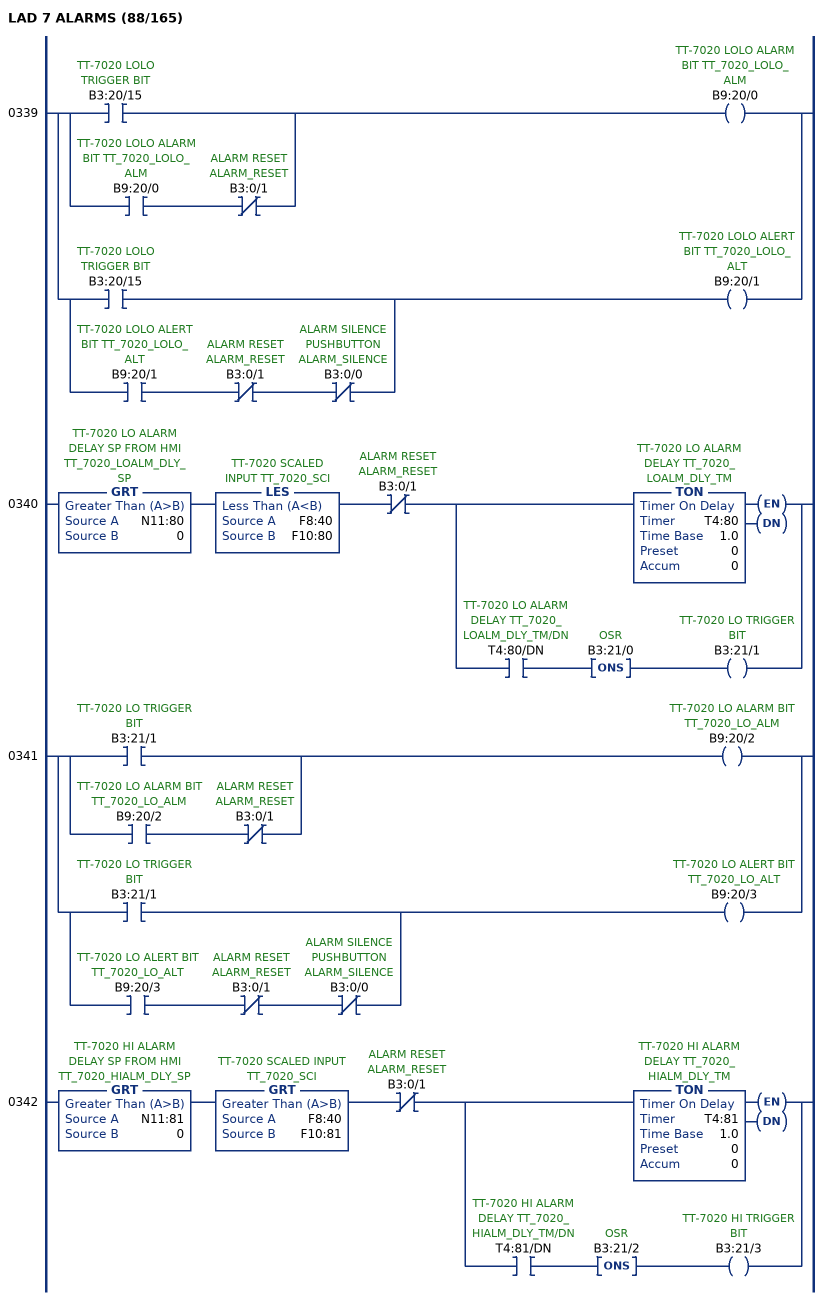
% Rung: 339 %
SOR BST BST XIC B3:20/15 NXB XIC B9:20/0 XIO B3:0/1 BND OTE B9:20/0 NXB BST XIC B3:20/15 NXB XIC B9:20/1 XIO B3:0/1 XIO B3:0/0 BND OTE B9:20/1 BND EOR
%   B3:20/15  "TT-7020 LOLO TRIGGER BIT" %
%   B9:20/0  TT_7020_LOLO_ALM  "TT-7020 LOLO ALARM BIT" %
%   B3:0/1  ALARM_RESET  "ALARM RESET" %
%   B9:20/1  TT_7020_LOLO_ALT  "TT-7020 LOLO ALERT BIT" %
%   B3:0/0  ALARM_SILENCE  "ALARM SILENCE PUSHBUTTON" %
% Rung: 340 %
SOR GRT N11:80 0 LES F8:40 F10:80 XIO B3:0/1 BST TON T4:80 1.0 0 0 NXB XIC T4:80/DN OSR B3:21/0 OTE B3:21/1 BND EOR
%   N11:80  TT_7020_LOALM_DLY_SP  "TT-7020 LO ALARM DELAY SP FROM HMI" %
%   F8:40  TT_7020_SCI  "TT-7020 SCALED INPUT" %
%   F10:80  TT_7020_LOALM_SP  "TT-7020 LO ALARM SP" %
%   B3:0/1  ALARM_RESET  "ALARM RESET" %
%   T4:80  TT_7020_LOALM_DLY_TM  "TT-7020 LO ALARM DELAY" %
%   B3:21/0  "OSR" %
%   B3:21/1  "TT-7020 LO TRIGGER BIT" %
% Rung: 341 %
SOR BST BST XIC B3:21/1 NXB XIC B9:20/2 XIO B3:0/1 BND OTE B9:20/2 NXB BST XIC B3:21/1 NXB XIC B9:20/3 XIO B3:0/1 XIO B3:0/0 BND OTE B9:20/3 BND EOR
%   B3:21/1  "TT-7020 LO TRIGGER BIT" %
%   B9:20/2  TT_7020_LO_ALM  "TT-7020 LO ALARM BIT" %
%   B3:0/1  ALARM_RESET  "ALARM RESET" %
%   B9:20/3  TT_7020_LO_ALT  "TT-7020 LO ALERT BIT" %
%   B3:0/0  ALARM_SILENCE  "ALARM SILENCE PUSHBUTTON" %
% Rung: 342 %
SOR GRT N11:81 0 GRT F8:40 F10:81 XIO B3:0/1 BST TON T4:81 1.0 0 0 NXB XIC T4:81/DN OSR B3:21/2 OTE B3:21/3 BND EOR
%   N11:81  TT_7020_HIALM_DLY_SP  "TT-7020 HI ALARM DELAY SP FROM HMI" %
%   F8:40  TT_7020_SCI  "TT-7020 SCALED INPUT" %
%   F10:81  TT_7020_HIALM_SP  "TT-7020 HI ALARM SP" %
%   B3:0/1  ALARM_RESET  "ALARM RESET" %
%   T4:81  TT_7020_HIALM_DLY_TM  "TT-7020 HI ALARM DELAY" %
%   B3:21/2  "OSR" %
%   B3:21/3  "TT-7020 HI TRIGGER BIT" %

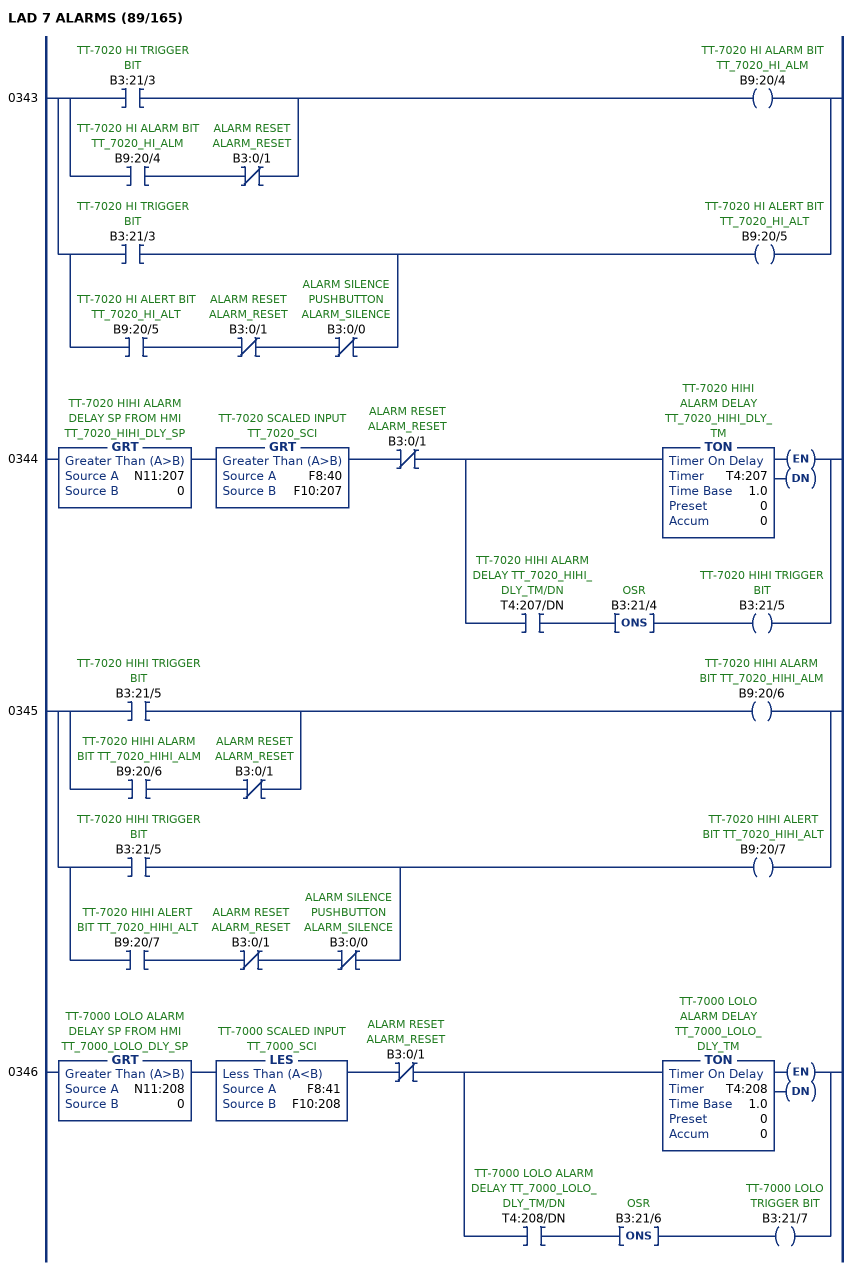
% Rung: 343 %
SOR BST BST XIC B3:21/3 NXB XIC B9:20/4 XIO B3:0/1 BND OTE B9:20/4 NXB BST XIC B3:21/3 NXB XIC B9:20/5 XIO B3:0/1 XIO B3:0/0 BND OTE B9:20/5 BND EOR
%   B3:21/3  "TT-7020 HI TRIGGER BIT" %
%   B9:20/4  TT_7020_HI_ALM  "TT-7020 HI ALARM BIT" %
%   B3:0/1  ALARM_RESET  "ALARM RESET" %
%   B9:20/5  TT_7020_HI_ALT  "TT-7020 HI ALERT BIT" %
%   B3:0/0  ALARM_SILENCE  "ALARM SILENCE PUSHBUTTON" %
% Rung: 344 %
SOR GRT N11:207 0 GRT F8:40 F10:207 XIO B3:0/1 BST TON T4:207 1.0 0 0 NXB XIC T4:207/DN OSR B3:21/4 OTE B3:21/5 BND EOR
%   N11:207  TT_7020_HIHI_DLY_SP  "TT-7020 HIHI ALARM DELAY SP FROM HMI" %
%   F8:40  TT_7020_SCI  "TT-7020 SCALED INPUT" %
%   F10:207  TT_7020_HIHI_SP  "TT-7020 HIHI ALARM SP" %
%   B3:0/1  ALARM_RESET  "ALARM RESET" %
%   T4:207  TT_7020_HIHI_DLY_TM  "TT-7020 HIHI ALARM DELAY" %
%   B3:21/4  "OSR" %
%   B3:21/5  "TT-7020 HIHI TRIGGER BIT" %
% Rung: 345 %
SOR BST BST XIC B3:21/5 NXB XIC B9:20/6 XIO B3:0/1 BND OTE B9:20/6 NXB BST XIC B3:21/5 NXB XIC B9:20/7 XIO B3:0/1 XIO B3:0/0 BND OTE B9:20/7 BND EOR
%   B3:21/5  "TT-7020 HIHI TRIGGER BIT" %
%   B9:20/6  TT_7020_HIHI_ALM  "TT-7020 HIHI ALARM BIT" %
%   B3:0/1  ALARM_RESET  "ALARM RESET" %
%   B9:20/7  TT_7020_HIHI_ALT  "TT-7020 HIHI ALERT BIT" %
%   B3:0/0  ALARM_SILENCE  "ALARM SILENCE PUSHBUTTON" %
% Rung: 346 %
SOR GRT N11:208 0 LES F8:41 F10:208 XIO B3:0/1 BST TON T4:208 1.0 0 0 NXB XIC T4:208/DN OSR B3:21/6 OTE B3:21/7 BND EOR
%   N11:208  TT_7000_LOLO_DLY_SP  "TT-7000 LOLO ALARM DELAY SP FROM HMI" %
%   F8:41  TT_7000_SCI  "TT-7000 SCALED INPUT" %
%   F10:208  TT_7000_LOLO_SP  "TT-7000 LOLO ALARM SP" %
%   B3:0/1  ALARM_RESET  "ALARM RESET" %
%   T4:208  TT_7000_LOLO_DLY_TM  "TT-7000 LOLO ALARM DELAY" %
%   B3:21/6  "OSR" %
%   B3:21/7  "TT-7000 LOLO TRIGGER BIT" %

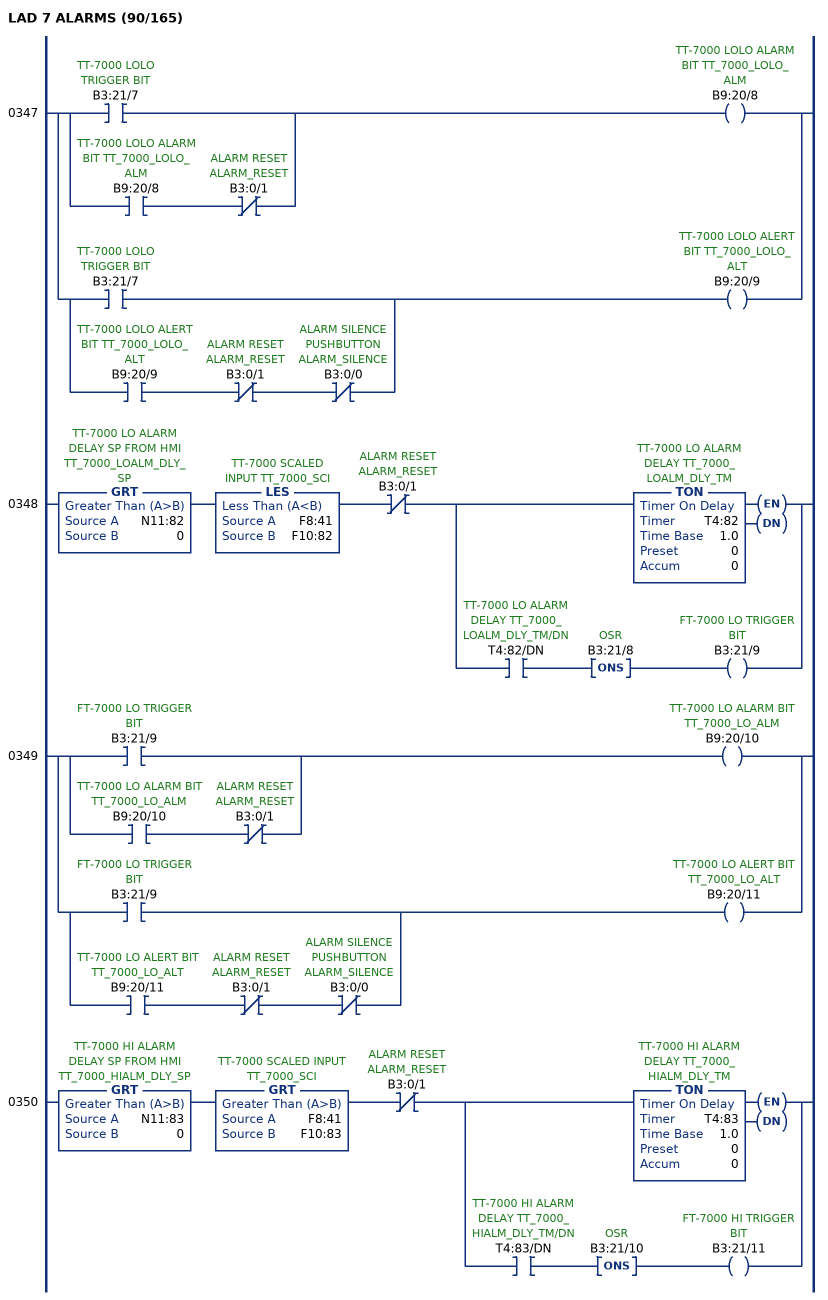
% Rung: 347 %
SOR BST BST XIC B3:21/7 NXB XIC B9:20/8 XIO B3:0/1 BND OTE B9:20/8 NXB BST XIC B3:21/7 NXB XIC B9:20/9 XIO B3:0/1 XIO B3:0/0 BND OTE B9:20/9 BND EOR
%   B3:21/7  "TT-7000 LOLO TRIGGER BIT" %
%   B9:20/8  TT_7000_LOLO_ALM  "TT-7000 LOLO ALARM BIT" %
%   B3:0/1  ALARM_RESET  "ALARM RESET" %
%   B9:20/9  TT_7000_LOLO_ALT  "TT-7000 LOLO ALERT BIT" %
%   B3:0/0  ALARM_SILENCE  "ALARM SILENCE PUSHBUTTON" %
% Rung: 348 %
SOR GRT N11:82 0 LES F8:41 F10:82 XIO B3:0/1 BST TON T4:82 1.0 0 0 NXB XIC T4:82/DN OSR B3:21/8 OTE B3:21/9 BND EOR
%   N11:82  TT_7000_LOALM_DLY_SP  "TT-7000 LO ALARM DELAY SP FROM HMI" %
%   F8:41  TT_7000_SCI  "TT-7000 SCALED INPUT" %
%   F10:82  TT_7000_LOALM_SP  "TT-7000 LO ALARM SP" %
%   B3:0/1  ALARM_RESET  "ALARM RESET" %
%   T4:82  TT_7000_LOALM_DLY_TM  "TT-7000 LO ALARM DELAY" %
%   B3:21/8  "OSR" %
%   B3:21/9  "FT-7000 LO TRIGGER BIT" %
% Rung: 349 %
SOR BST BST XIC B3:21/9 NXB XIC B9:20/10 XIO B3:0/1 BND OTE B9:20/10 NXB BST XIC B3:21/9 NXB XIC B9:20/11 XIO B3:0/1 XIO B3:0/0 BND OTE B9:20/11 BND EOR
%   B3:21/9  "FT-7000 LO TRIGGER BIT" %
%   B9:20/10  TT_7000_LO_ALM  "TT-7000 LO ALARM BIT" %
%   B3:0/1  ALARM_RESET  "ALARM RESET" %
%   B9:20/11  TT_7000_LO_ALT  "TT-7000 LO ALERT BIT" %
%   B3:0/0  ALARM_SILENCE  "ALARM SILENCE PUSHBUTTON" %
% Rung: 350 %
SOR GRT N11:83 0 GRT F8:41 F10:83 XIO B3:0/1 BST TON T4:83 1.0 0 0 NXB XIC T4:83/DN OSR B3:21/10 OTE B3:21/11 BND EOR
%   N11:83  TT_7000_HIALM_DLY_SP  "TT-7000 HI ALARM DELAY SP FROM HMI" %
%   F8:41  TT_7000_SCI  "TT-7000 SCALED INPUT" %
%   F10:83  TT_7000_HIALM_SP  "TT-7000 HI ALARM SP" %
%   B3:0/1  ALARM_RESET  "ALARM RESET" %
%   T4:83  TT_7000_HIALM_DLY_TM  "TT-7000 HI ALARM DELAY" %
%   B3:21/10  "OSR" %
%   B3:21/11  "FT-7000 HI TRIGGER BIT" %

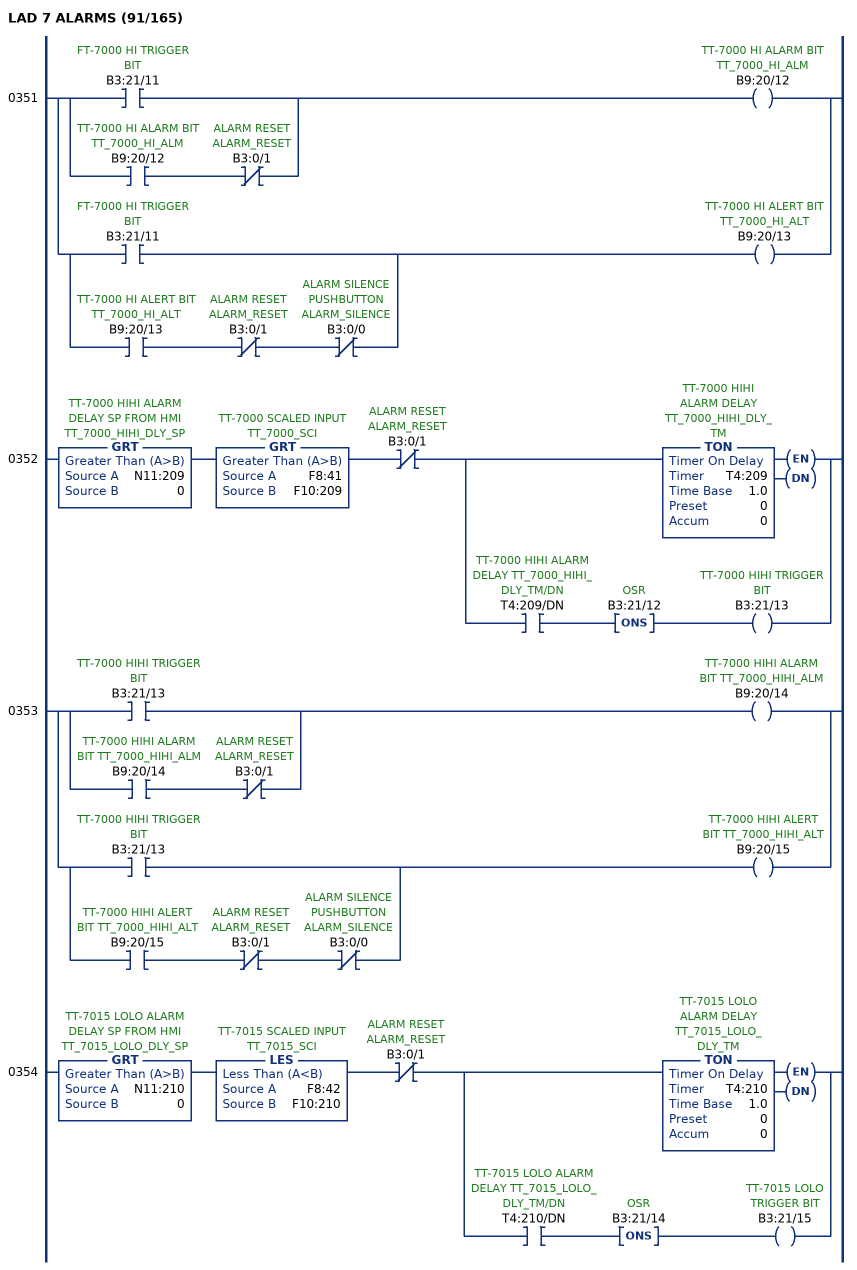
% Rung: 351 %
SOR BST BST XIC B3:21/11 NXB XIC B9:20/12 XIO B3:0/1 BND OTE B9:20/12 NXB BST XIC B3:21/11 NXB XIC B9:20/13 XIO B3:0/1 XIO B3:0/0 BND OTE B9:20/13 BND EOR
%   B3:21/11  "FT-7000 HI TRIGGER BIT" %
%   B9:20/12  TT_7000_HI_ALM  "TT-7000 HI ALARM BIT" %
%   B3:0/1  ALARM_RESET  "ALARM RESET" %
%   B9:20/13  TT_7000_HI_ALT  "TT-7000 HI ALERT BIT" %
%   B3:0/0  ALARM_SILENCE  "ALARM SILENCE PUSHBUTTON" %
% Rung: 352 %
SOR GRT N11:209 0 GRT F8:41 F10:209 XIO B3:0/1 BST TON T4:209 1.0 0 0 NXB XIC T4:209/DN OSR B3:21/12 OTE B3:21/13 BND EOR
%   N11:209  TT_7000_HIHI_DLY_SP  "TT-7000 HIHI ALARM DELAY SP FROM HMI" %
%   F8:41  TT_7000_SCI  "TT-7000 SCALED INPUT" %
%   F10:209  TT_7000_HIHI_SP  "TT-7000 HIHI ALARM SP" %
%   B3:0/1  ALARM_RESET  "ALARM RESET" %
%   T4:209  TT_7000_HIHI_DLY_TM  "TT-7000 HIHI ALARM DELAY" %
%   B3:21/12  "OSR" %
%   B3:21/13  "TT-7000 HIHI TRIGGER BIT" %
% Rung: 353 %
SOR BST BST XIC B3:21/13 NXB XIC B9:20/14 XIO B3:0/1 BND OTE B9:20/14 NXB BST XIC B3:21/13 NXB XIC B9:20/15 XIO B3:0/1 XIO B3:0/0 BND OTE B9:20/15 BND EOR
%   B3:21/13  "TT-7000 HIHI TRIGGER BIT" %
%   B9:20/14  TT_7000_HIHI_ALM  "TT-7000 HIHI ALARM BIT" %
%   B3:0/1  ALARM_RESET  "ALARM RESET" %
%   B9:20/15  TT_7000_HIHI_ALT  "TT-7000 HIHI ALERT BIT" %
%   B3:0/0  ALARM_SILENCE  "ALARM SILENCE PUSHBUTTON" %
% Rung: 354 %
SOR GRT N11:210 0 LES F8:42 F10:210 XIO B3:0/1 BST TON T4:210 1.0 0 0 NXB XIC T4:210/DN OSR B3:21/14 OTE B3:21/15 BND EOR
%   N11:210  TT_7015_LOLO_DLY_SP  "TT-7015 LOLO ALARM DELAY SP FROM HMI" %
%   F8:42  TT_7015_SCI  "TT-7015 SCALED INPUT" %
%   F10:210  TT_7015_LOLO_SP  "TT-7015 LOLO ALARM SP" %
%   B3:0/1  ALARM_RESET  "ALARM RESET" %
%   T4:210  TT_7015_LOLO_DLY_TM  "TT-7015 LOLO ALARM DELAY" %
%   B3:21/14  "OSR" %
%   B3:21/15  "TT-7015 LOLO TRIGGER BIT" %

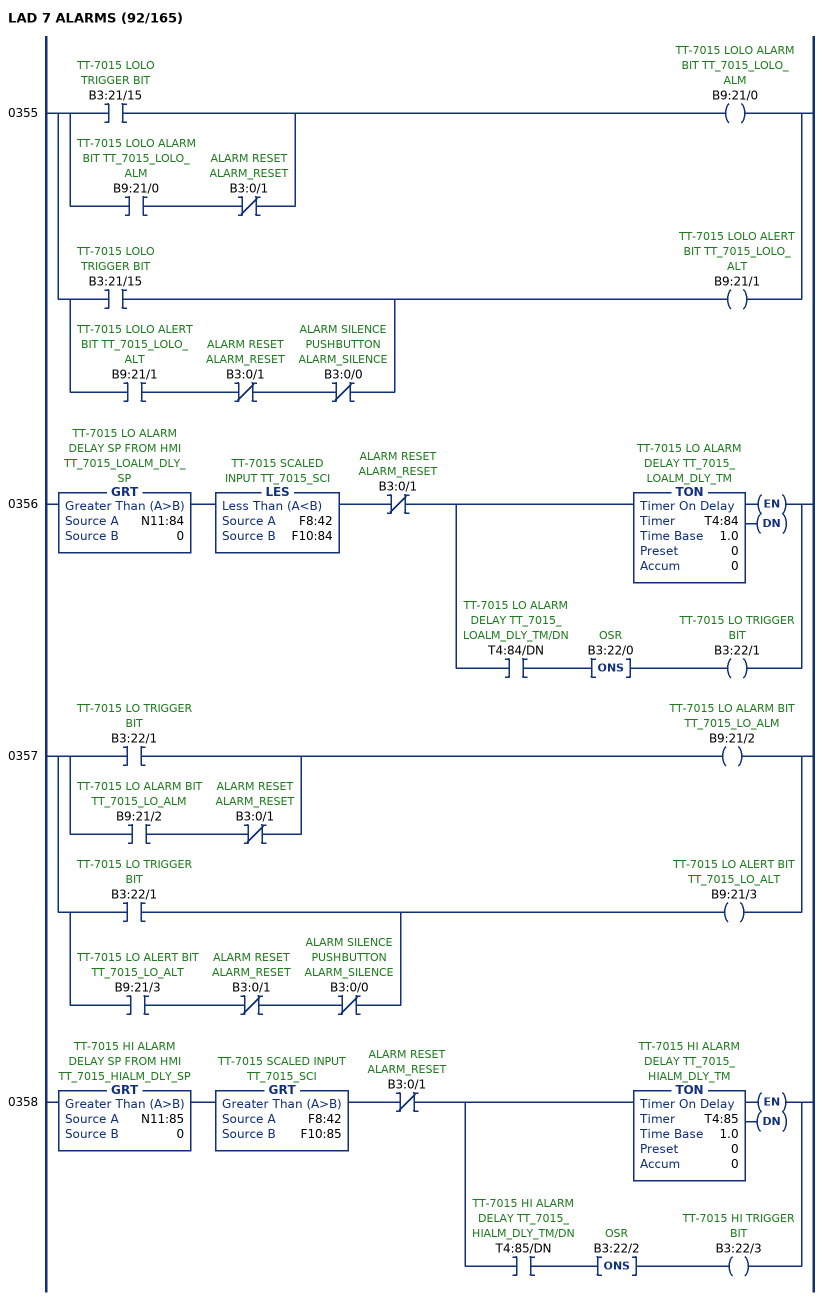
% Rung: 355 %
SOR BST BST XIC B3:21/15 NXB XIC B9:21/0 XIO B3:0/1 BND OTE B9:21/0 NXB BST XIC B3:21/15 NXB XIC B9:21/1 XIO B3:0/1 XIO B3:0/0 BND OTE B9:21/1 BND EOR
%   B3:21/15  "TT-7015 LOLO TRIGGER BIT" %
%   B9:21/0  TT_7015_LOLO_ALM  "TT-7015 LOLO ALARM BIT" %
%   B3:0/1  ALARM_RESET  "ALARM RESET" %
%   B9:21/1  TT_7015_LOLO_ALT  "TT-7015 LOLO ALERT BIT" %
%   B3:0/0  ALARM_SILENCE  "ALARM SILENCE PUSHBUTTON" %
% Rung: 356 %
SOR GRT N11:84 0 LES F8:42 F10:84 XIO B3:0/1 BST TON T4:84 1.0 0 0 NXB XIC T4:84/DN OSR B3:22/0 OTE B3:22/1 BND EOR
%   N11:84  TT_7015_LOALM_DLY_SP  "TT-7015 LO ALARM DELAY SP FROM HMI" %
%   F8:42  TT_7015_SCI  "TT-7015 SCALED INPUT" %
%   F10:84  TT_7015_LOALM_SP  "TT-7015 LO ALARM SP" %
%   B3:0/1  ALARM_RESET  "ALARM RESET" %
%   T4:84  TT_7015_LOALM_DLY_TM  "TT-7015 LO ALARM DELAY" %
%   B3:22/0  "OSR" %
%   B3:22/1  "TT-7015 LO TRIGGER BIT" %
% Rung: 357 %
SOR BST BST XIC B3:22/1 NXB XIC B9:21/2 XIO B3:0/1 BND OTE B9:21/2 NXB BST XIC B3:22/1 NXB XIC B9:21/3 XIO B3:0/1 XIO B3:0/0 BND OTE B9:21/3 BND EOR
%   B3:22/1  "TT-7015 LO TRIGGER BIT" %
%   B9:21/2  TT_7015_LO_ALM  "TT-7015 LO ALARM BIT" %
%   B3:0/1  ALARM_RESET  "ALARM RESET" %
%   B9:21/3  TT_7015_LO_ALT  "TT-7015 LO ALERT BIT" %
%   B3:0/0  ALARM_SILENCE  "ALARM SILENCE PUSHBUTTON" %
% Rung: 358 %
SOR GRT N11:85 0 GRT F8:42 F10:85 XIO B3:0/1 BST TON T4:85 1.0 0 0 NXB XIC T4:85/DN OSR B3:22/2 OTE B3:22/3 BND EOR
%   N11:85  TT_7015_HIALM_DLY_SP  "TT-7015 HI ALARM DELAY SP FROM HMI" %
%   F8:42  TT_7015_SCI  "TT-7015 SCALED INPUT" %
%   F10:85  TT_7015_HIALM_SP  "TT-7015 HI ALARM SP" %
%   B3:0/1  ALARM_RESET  "ALARM RESET" %
%   T4:85  TT_7015_HIALM_DLY_TM  "TT-7015 HI ALARM DELAY" %
%   B3:22/2  "OSR" %
%   B3:22/3  "TT-7015 HI TRIGGER BIT" %

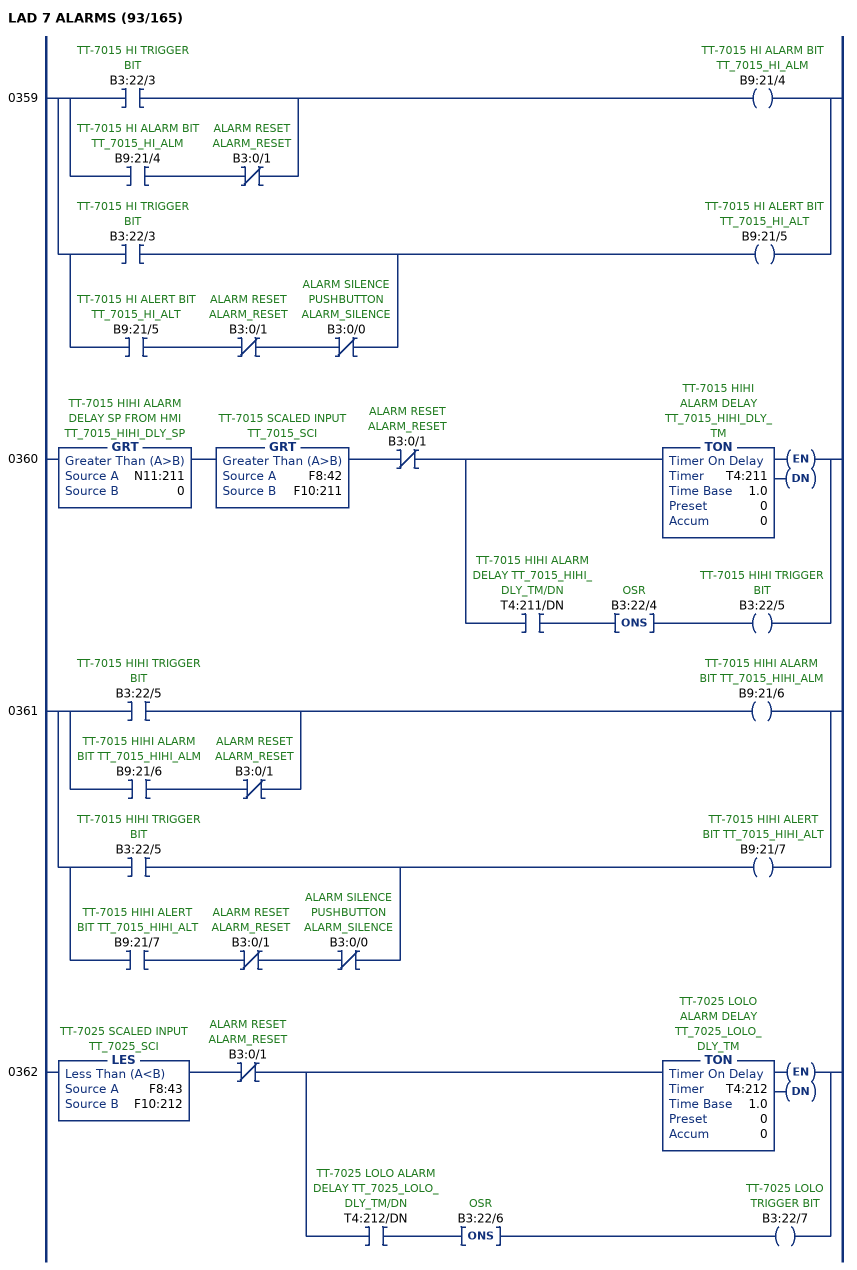
% Rung: 359 %
SOR BST BST XIC B3:22/3 NXB XIC B9:21/4 XIO B3:0/1 BND OTE B9:21/4 NXB BST XIC B3:22/3 NXB XIC B9:21/5 XIO B3:0/1 XIO B3:0/0 BND OTE B9:21/5 BND EOR
%   B3:22/3  "TT-7015 HI TRIGGER BIT" %
%   B9:21/4  TT_7015_HI_ALM  "TT-7015 HI ALARM BIT" %
%   B3:0/1  ALARM_RESET  "ALARM RESET" %
%   B9:21/5  TT_7015_HI_ALT  "TT-7015 HI ALERT BIT" %
%   B3:0/0  ALARM_SILENCE  "ALARM SILENCE PUSHBUTTON" %
% Rung: 360 %
SOR GRT N11:211 0 GRT F8:42 F10:211 XIO B3:0/1 BST TON T4:211 1.0 0 0 NXB XIC T4:211/DN OSR B3:22/4 OTE B3:22/5 BND EOR
%   N11:211  TT_7015_HIHI_DLY_SP  "TT-7015 HIHI ALARM DELAY SP FROM HMI" %
%   F8:42  TT_7015_SCI  "TT-7015 SCALED INPUT" %
%   F10:211  TT_7015_HIHI_SP  "TT-7015 HIHI ALARM SP" %
%   B3:0/1  ALARM_RESET  "ALARM RESET" %
%   T4:211  TT_7015_HIHI_DLY_TM  "TT-7015 HIHI ALARM DELAY" %
%   B3:22/4  "OSR" %
%   B3:22/5  "TT-7015 HIHI TRIGGER BIT" %
% Rung: 361 %
SOR BST BST XIC B3:22/5 NXB XIC B9:21/6 XIO B3:0/1 BND OTE B9:21/6 NXB BST XIC B3:22/5 NXB XIC B9:21/7 XIO B3:0/1 XIO B3:0/0 BND OTE B9:21/7 BND EOR
%   B3:22/5  "TT-7015 HIHI TRIGGER BIT" %
%   B9:21/6  TT_7015_HIHI_ALM  "TT-7015 HIHI ALARM BIT" %
%   B3:0/1  ALARM_RESET  "ALARM RESET" %
%   B9:21/7  TT_7015_HIHI_ALT  "TT-7015 HIHI ALERT BIT" %
%   B3:0/0  ALARM_SILENCE  "ALARM SILENCE PUSHBUTTON" %
% Rung: 362 %
SOR LES F8:43 F10:212 XIO B3:0/1 BST TON T4:212 1.0 0 0 NXB XIC T4:212/DN OSR B3:22/6 OTE B3:22/7 BND EOR
%   F8:43  TT_7025_SCI  "TT-7025 SCALED INPUT" %
%   F10:212  TT_7025_LOLO_SP  "TT-7025 LOLO ALARM SP" %
%   B3:0/1  ALARM_RESET  "ALARM RESET" %
%   T4:212  TT_7025_LOLO_DLY_TM  "TT-7025 LOLO ALARM DELAY" %
%   B3:22/6  "OSR" %
%   B3:22/7  "TT-7025 LOLO TRIGGER BIT" %

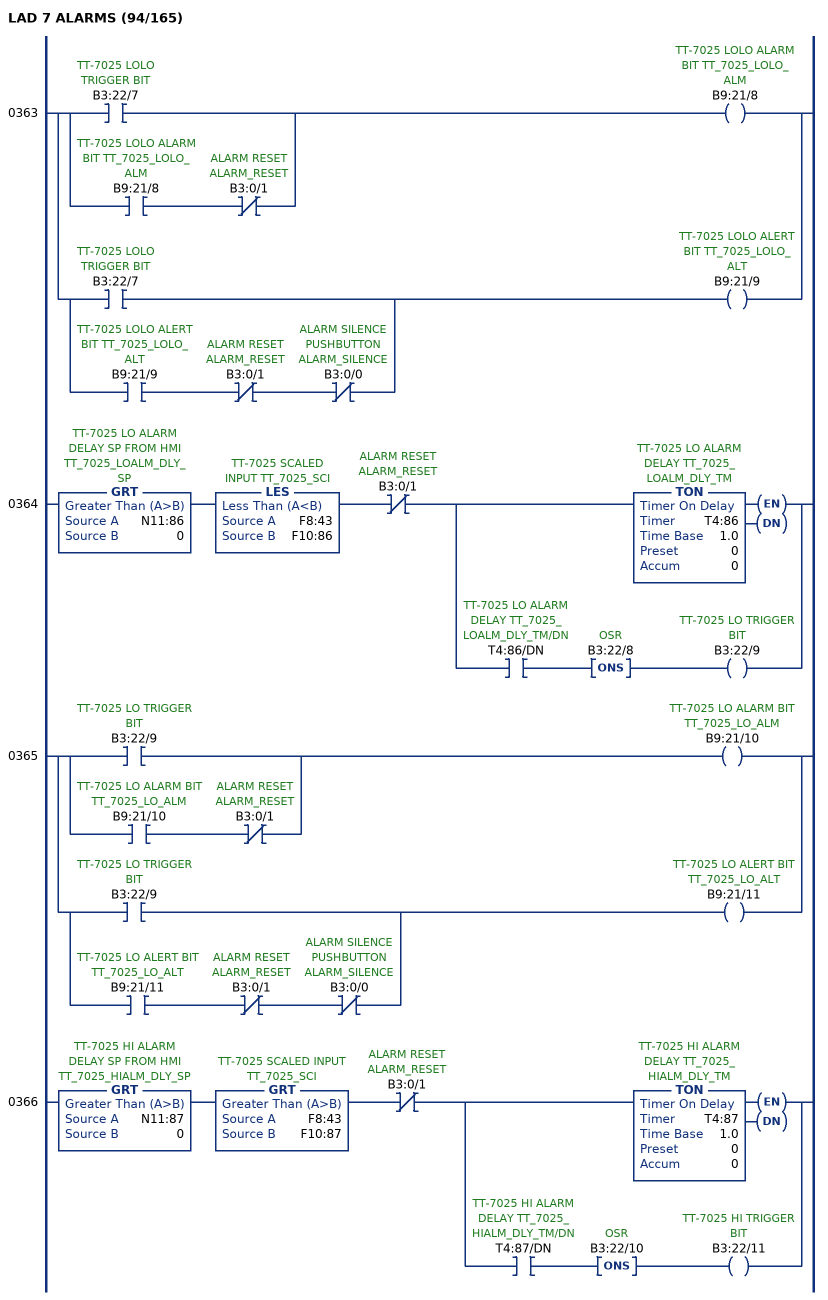
% Rung: 363 %
SOR BST BST XIC B3:22/7 NXB XIC B9:21/8 XIO B3:0/1 BND OTE B9:21/8 NXB BST XIC B3:22/7 NXB XIC B9:21/9 XIO B3:0/1 XIO B3:0/0 BND OTE B9:21/9 BND EOR
%   B3:22/7  "TT-7025 LOLO TRIGGER BIT" %
%   B9:21/8  TT_7025_LOLO_ALM  "TT-7025 LOLO ALARM BIT" %
%   B3:0/1  ALARM_RESET  "ALARM RESET" %
%   B9:21/9  TT_7025_LOLO_ALT  "TT-7025 LOLO ALERT BIT" %
%   B3:0/0  ALARM_SILENCE  "ALARM SILENCE PUSHBUTTON" %
% Rung: 364 %
SOR GRT N11:86 0 LES F8:43 F10:86 XIO B3:0/1 BST TON T4:86 1.0 0 0 NXB XIC T4:86/DN OSR B3:22/8 OTE B3:22/9 BND EOR
%   N11:86  TT_7025_LOALM_DLY_SP  "TT-7025 LO ALARM DELAY SP FROM HMI" %
%   F8:43  TT_7025_SCI  "TT-7025 SCALED INPUT" %
%   F10:86  TT_7025_LOALM_SP  "TT-7025 LO ALARM SP" %
%   B3:0/1  ALARM_RESET  "ALARM RESET" %
%   T4:86  TT_7025_LOALM_DLY_TM  "TT-7025 LO ALARM DELAY" %
%   B3:22/8  "OSR" %
%   B3:22/9  "TT-7025 LO TRIGGER BIT" %
% Rung: 365 %
SOR BST BST XIC B3:22/9 NXB XIC B9:21/10 XIO B3:0/1 BND OTE B9:21/10 NXB BST XIC B3:22/9 NXB XIC B9:21/11 XIO B3:0/1 XIO B3:0/0 BND OTE B9:21/11 BND EOR
%   B3:22/9  "TT-7025 LO TRIGGER BIT" %
%   B9:21/10  TT_7025_LO_ALM  "TT-7025 LO ALARM BIT" %
%   B3:0/1  ALARM_RESET  "ALARM RESET" %
%   B9:21/11  TT_7025_LO_ALT  "TT-7025 LO ALERT BIT" %
%   B3:0/0  ALARM_SILENCE  "ALARM SILENCE PUSHBUTTON" %
% Rung: 366 %
SOR GRT N11:87 0 GRT F8:43 F10:87 XIO B3:0/1 BST TON T4:87 1.0 0 0 NXB XIC T4:87/DN OSR B3:22/10 OTE B3:22/11 BND EOR
%   N11:87  TT_7025_HIALM_DLY_SP  "TT-7025 HI ALARM DELAY SP FROM HMI" %
%   F8:43  TT_7025_SCI  "TT-7025 SCALED INPUT" %
%   F10:87  TT_7025_HIALM_SP  "TT-7025 HI ALARM SP" %
%   B3:0/1  ALARM_RESET  "ALARM RESET" %
%   T4:87  TT_7025_HIALM_DLY_TM  "TT-7025 HI ALARM DELAY" %
%   B3:22/10  "OSR" %
%   B3:22/11  "TT-7025 HI TRIGGER BIT" %

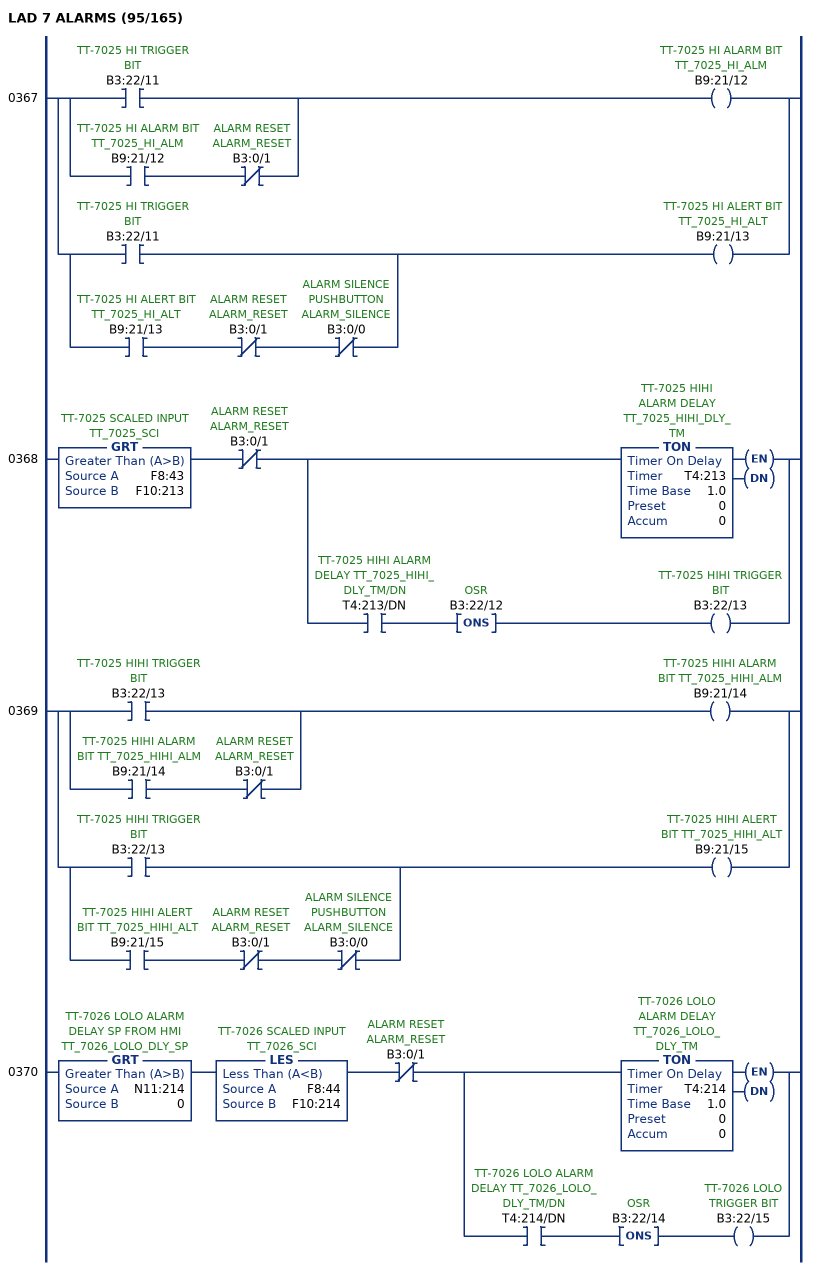
% Rung: 367 %
SOR BST BST XIC B3:22/11 NXB XIC B9:21/12 XIO B3:0/1 BND OTE B9:21/12 NXB BST XIC B3:22/11 NXB XIC B9:21/13 XIO B3:0/1 XIO B3:0/0 BND OTE B9:21/13 BND EOR
%   B3:22/11  "TT-7025 HI TRIGGER BIT" %
%   B9:21/12  TT_7025_HI_ALM  "TT-7025 HI ALARM BIT" %
%   B3:0/1  ALARM_RESET  "ALARM RESET" %
%   B9:21/13  TT_7025_HI_ALT  "TT-7025 HI ALERT BIT" %
%   B3:0/0  ALARM_SILENCE  "ALARM SILENCE PUSHBUTTON" %
% Rung: 368 %
SOR GRT F8:43 F10:213 XIO B3:0/1 BST TON T4:213 1.0 0 0 NXB XIC T4:213/DN OSR B3:22/12 OTE B3:22/13 BND EOR
%   F8:43  TT_7025_SCI  "TT-7025 SCALED INPUT" %
%   F10:213  TT_7025_HIHI_SP  "TT-7025 HIHI ALARM SP" %
%   B3:0/1  ALARM_RESET  "ALARM RESET" %
%   T4:213  TT_7025_HIHI_DLY_TM  "TT-7025 HIHI ALARM DELAY" %
%   B3:22/12  "OSR" %
%   B3:22/13  "TT-7025 HIHI TRIGGER BIT" %
% Rung: 369 %
SOR BST BST XIC B3:22/13 NXB XIC B9:21/14 XIO B3:0/1 BND OTE B9:21/14 NXB BST XIC B3:22/13 NXB XIC B9:21/15 XIO B3:0/1 XIO B3:0/0 BND OTE B9:21/15 BND EOR
%   B3:22/13  "TT-7025 HIHI TRIGGER BIT" %
%   B9:21/14  TT_7025_HIHI_ALM  "TT-7025 HIHI ALARM BIT" %
%   B3:0/1  ALARM_RESET  "ALARM RESET" %
%   B9:21/15  TT_7025_HIHI_ALT  "TT-7025 HIHI ALERT BIT" %
%   B3:0/0  ALARM_SILENCE  "ALARM SILENCE PUSHBUTTON" %
% Rung: 370 %
SOR GRT N11:214 0 LES F8:44 F10:214 XIO B3:0/1 BST TON T4:214 1.0 0 0 NXB XIC T4:214/DN OSR B3:22/14 OTE B3:22/15 BND EOR
%   N11:214  TT_7026_LOLO_DLY_SP  "TT-7026 LOLO ALARM DELAY SP FROM HMI" %
%   F8:44  TT_7026_SCI  "TT-7026 SCALED INPUT" %
%   F10:214  TT_7026_LOLO_SP  "TT-7026 LOLO ALARM SP" %
%   B3:0/1  ALARM_RESET  "ALARM RESET" %
%   T4:214  TT_7026_LOLO_DLY_TM  "TT-7026 LOLO ALARM DELAY" %
%   B3:22/14  "OSR" %
%   B3:22/15  "TT-7026 LOLO TRIGGER BIT" %

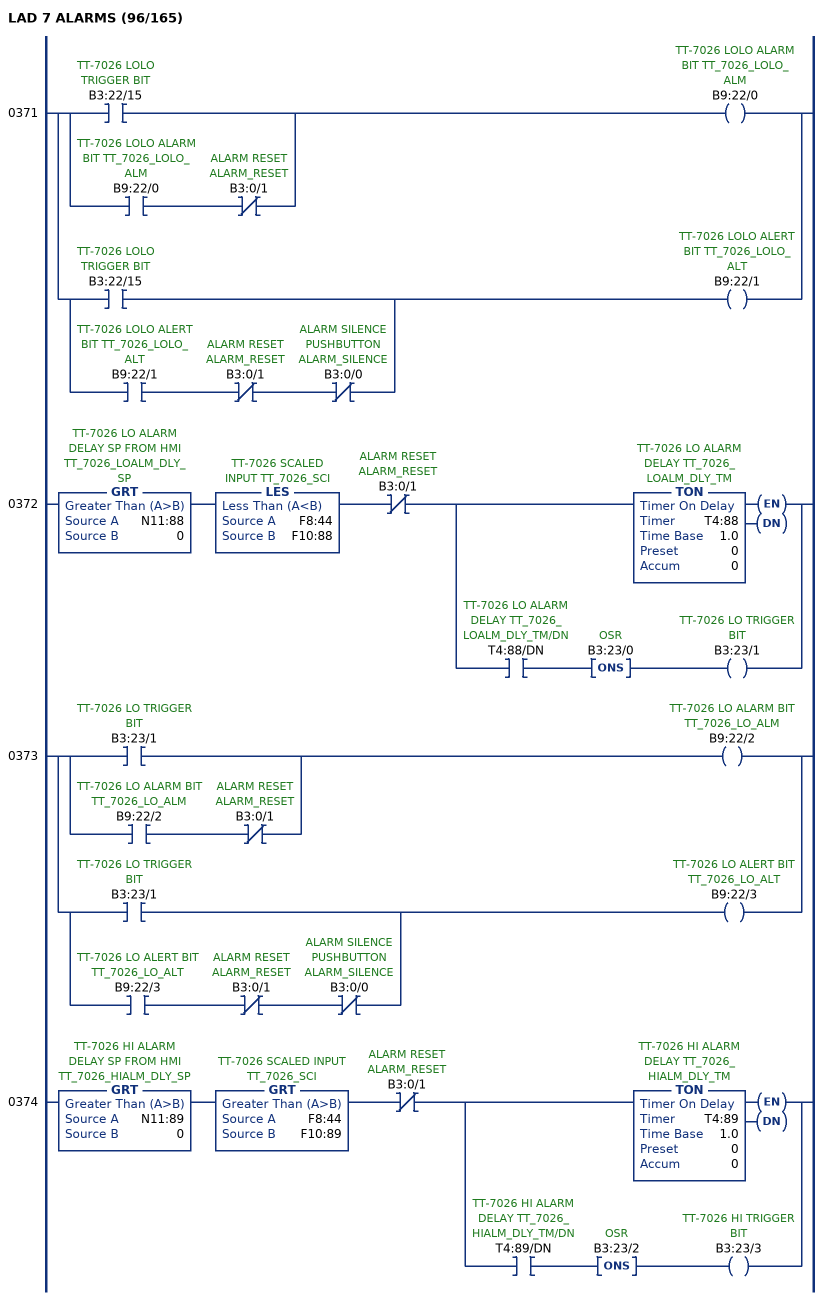
% Rung: 371 %
SOR BST BST XIC B3:22/15 NXB XIC B9:22/0 XIO B3:0/1 BND OTE B9:22/0 NXB BST XIC B3:22/15 NXB XIC B9:22/1 XIO B3:0/1 XIO B3:0/0 BND OTE B9:22/1 BND EOR
%   B3:22/15  "TT-7026 LOLO TRIGGER BIT" %
%   B9:22/0  TT_7026_LOLO_ALM  "TT-7026 LOLO ALARM BIT" %
%   B3:0/1  ALARM_RESET  "ALARM RESET" %
%   B9:22/1  TT_7026_LOLO_ALT  "TT-7026 LOLO ALERT BIT" %
%   B3:0/0  ALARM_SILENCE  "ALARM SILENCE PUSHBUTTON" %
% Rung: 372 %
SOR GRT N11:88 0 LES F8:44 F10:88 XIO B3:0/1 BST TON T4:88 1.0 0 0 NXB XIC T4:88/DN OSR B3:23/0 OTE B3:23/1 BND EOR
%   N11:88  TT_7026_LOALM_DLY_SP  "TT-7026 LO ALARM DELAY SP FROM HMI" %
%   F8:44  TT_7026_SCI  "TT-7026 SCALED INPUT" %
%   F10:88  TT_7026_LOALM_SP  "TT-7026 LO ALARM SP" %
%   B3:0/1  ALARM_RESET  "ALARM RESET" %
%   T4:88  TT_7026_LOALM_DLY_TM  "TT-7026 LO ALARM DELAY" %
%   B3:23/0  "OSR" %
%   B3:23/1  "TT-7026 LO TRIGGER BIT" %
% Rung: 373 %
SOR BST BST XIC B3:23/1 NXB XIC B9:22/2 XIO B3:0/1 BND OTE B9:22/2 NXB BST XIC B3:23/1 NXB XIC B9:22/3 XIO B3:0/1 XIO B3:0/0 BND OTE B9:22/3 BND EOR
%   B3:23/1  "TT-7026 LO TRIGGER BIT" %
%   B9:22/2  TT_7026_LO_ALM  "TT-7026 LO ALARM BIT" %
%   B3:0/1  ALARM_RESET  "ALARM RESET" %
%   B9:22/3  TT_7026_LO_ALT  "TT-7026 LO ALERT BIT" %
%   B3:0/0  ALARM_SILENCE  "ALARM SILENCE PUSHBUTTON" %
% Rung: 374 %
SOR GRT N11:89 0 GRT F8:44 F10:89 XIO B3:0/1 BST TON T4:89 1.0 0 0 NXB XIC T4:89/DN OSR B3:23/2 OTE B3:23/3 BND EOR
%   N11:89  TT_7026_HIALM_DLY_SP  "TT-7026 HI ALARM DELAY SP FROM HMI" %
%   F8:44  TT_7026_SCI  "TT-7026 SCALED INPUT" %
%   F10:89  TT_7026_HIALM_SP  "TT-7026 HI ALARM SP" %
%   B3:0/1  ALARM_RESET  "ALARM RESET" %
%   T4:89  TT_7026_HIALM_DLY_TM  "TT-7026 HI ALARM DELAY" %
%   B3:23/2  "OSR" %
%   B3:23/3  "TT-7026 HI TRIGGER BIT" %

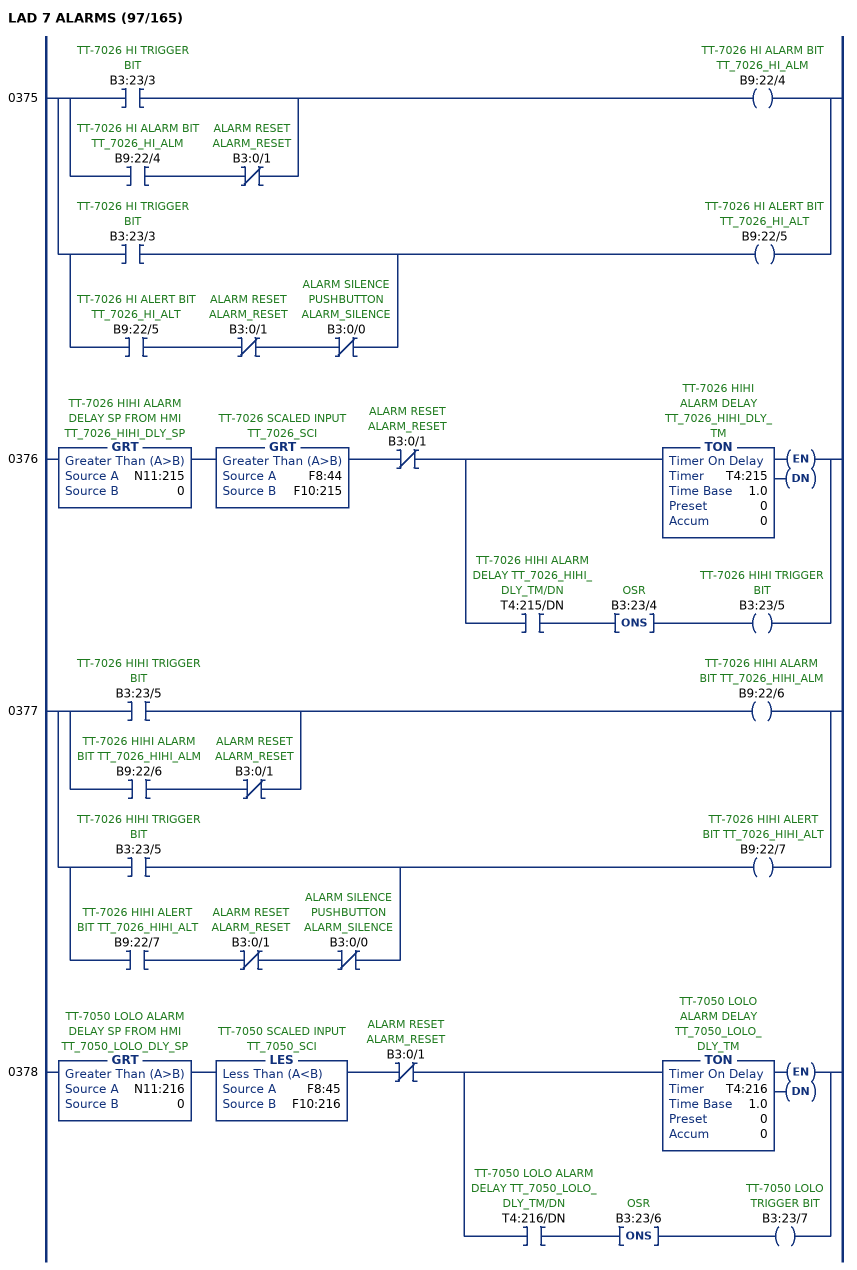
% Rung: 375 %
SOR BST BST XIC B3:23/3 NXB XIC B9:22/4 XIO B3:0/1 BND OTE B9:22/4 NXB BST XIC B3:23/3 NXB XIC B9:22/5 XIO B3:0/1 XIO B3:0/0 BND OTE B9:22/5 BND EOR
%   B3:23/3  "TT-7026 HI TRIGGER BIT" %
%   B9:22/4  TT_7026_HI_ALM  "TT-7026 HI ALARM BIT" %
%   B3:0/1  ALARM_RESET  "ALARM RESET" %
%   B9:22/5  TT_7026_HI_ALT  "TT-7026 HI ALERT BIT" %
%   B3:0/0  ALARM_SILENCE  "ALARM SILENCE PUSHBUTTON" %
% Rung: 376 %
SOR GRT N11:215 0 GRT F8:44 F10:215 XIO B3:0/1 BST TON T4:215 1.0 0 0 NXB XIC T4:215/DN OSR B3:23/4 OTE B3:23/5 BND EOR
%   N11:215  TT_7026_HIHI_DLY_SP  "TT-7026 HIHI ALARM DELAY SP FROM HMI" %
%   F8:44  TT_7026_SCI  "TT-7026 SCALED INPUT" %
%   F10:215  TT_7026_HIHI_SP  "TT-7026 HIHI ALARM SP" %
%   B3:0/1  ALARM_RESET  "ALARM RESET" %
%   T4:215  TT_7026_HIHI_DLY_TM  "TT-7026 HIHI ALARM DELAY" %
%   B3:23/4  "OSR" %
%   B3:23/5  "TT-7026 HIHI TRIGGER BIT" %
% Rung: 377 %
SOR BST BST XIC B3:23/5 NXB XIC B9:22/6 XIO B3:0/1 BND OTE B9:22/6 NXB BST XIC B3:23/5 NXB XIC B9:22/7 XIO B3:0/1 XIO B3:0/0 BND OTE B9:22/7 BND EOR
%   B3:23/5  "TT-7026 HIHI TRIGGER BIT" %
%   B9:22/6  TT_7026_HIHI_ALM  "TT-7026 HIHI ALARM BIT" %
%   B3:0/1  ALARM_RESET  "ALARM RESET" %
%   B9:22/7  TT_7026_HIHI_ALT  "TT-7026 HIHI ALERT BIT" %
%   B3:0/0  ALARM_SILENCE  "ALARM SILENCE PUSHBUTTON" %
% Rung: 378 %
SOR GRT N11:216 0 LES F8:45 F10:216 XIO B3:0/1 BST TON T4:216 1.0 0 0 NXB XIC T4:216/DN OSR B3:23/6 OTE B3:23/7 BND EOR
%   N11:216  TT_7050_LOLO_DLY_SP  "TT-7050 LOLO ALARM DELAY SP FROM HMI" %
%   F8:45  TT_7050_SCI  "TT-7050 SCALED INPUT" %
%   F10:216  TT_7050_LOLO_SP  "TT-7050 LOLO ALARM SP" %
%   B3:0/1  ALARM_RESET  "ALARM RESET" %
%   T4:216  TT_7050_LOLO_DLY_TM  "TT-7050 LOLO ALARM DELAY" %
%   B3:23/6  "OSR" %
%   B3:23/7  "TT-7050 LOLO TRIGGER BIT" %

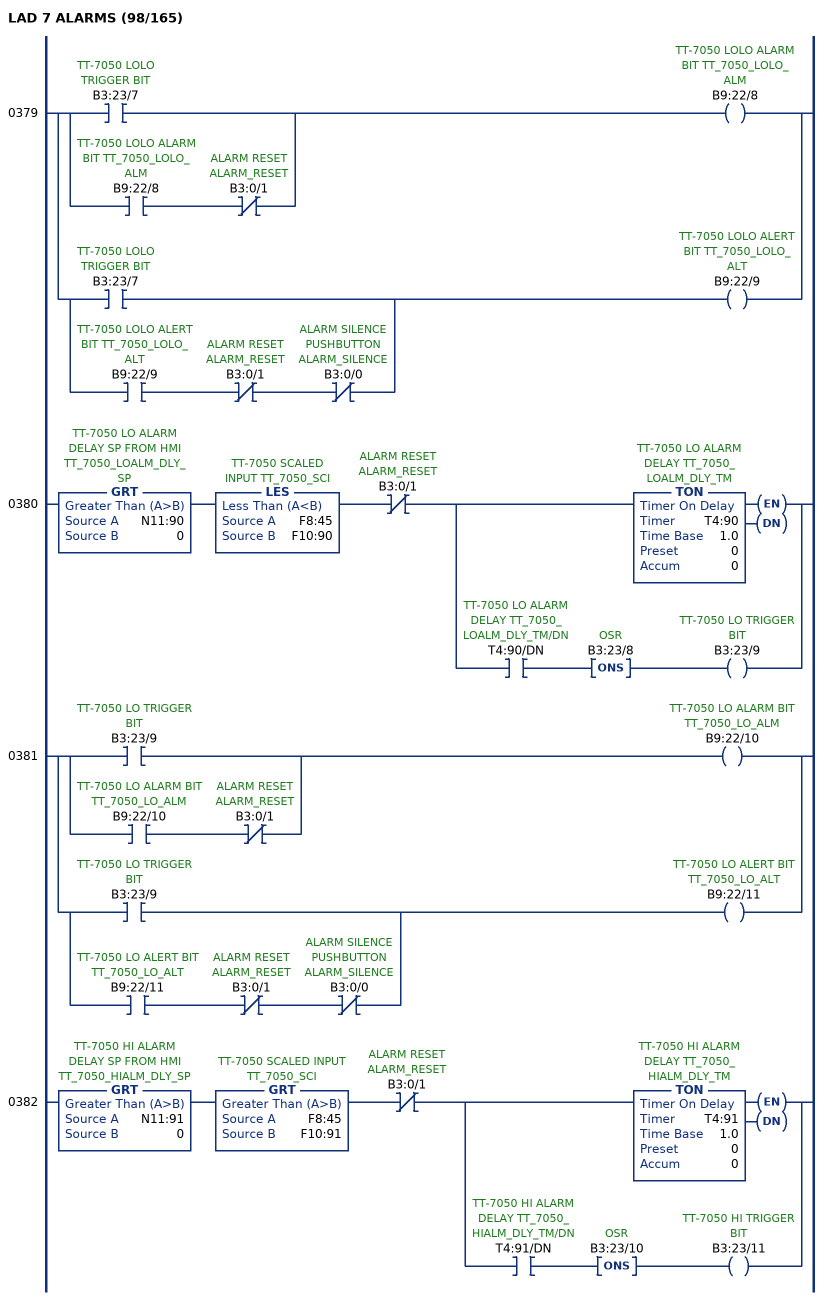
% Rung: 379 %
SOR BST BST XIC B3:23/7 NXB XIC B9:22/8 XIO B3:0/1 BND OTE B9:22/8 NXB BST XIC B3:23/7 NXB XIC B9:22/9 XIO B3:0/1 XIO B3:0/0 BND OTE B9:22/9 BND EOR
%   B3:23/7  "TT-7050 LOLO TRIGGER BIT" %
%   B9:22/8  TT_7050_LOLO_ALM  "TT-7050 LOLO ALARM BIT" %
%   B3:0/1  ALARM_RESET  "ALARM RESET" %
%   B9:22/9  TT_7050_LOLO_ALT  "TT-7050 LOLO ALERT BIT" %
%   B3:0/0  ALARM_SILENCE  "ALARM SILENCE PUSHBUTTON" %
% Rung: 380 %
SOR GRT N11:90 0 LES F8:45 F10:90 XIO B3:0/1 BST TON T4:90 1.0 0 0 NXB XIC T4:90/DN OSR B3:23/8 OTE B3:23/9 BND EOR
%   N11:90  TT_7050_LOALM_DLY_SP  "TT-7050 LO ALARM DELAY SP FROM HMI" %
%   F8:45  TT_7050_SCI  "TT-7050 SCALED INPUT" %
%   F10:90  TT_7050_LOALM_SP  "TT-7050 LO ALARM SP" %
%   B3:0/1  ALARM_RESET  "ALARM RESET" %
%   T4:90  TT_7050_LOALM_DLY_TM  "TT-7050 LO ALARM DELAY" %
%   B3:23/8  "OSR" %
%   B3:23/9  "TT-7050 LO TRIGGER BIT" %
% Rung: 381 %
SOR BST BST XIC B3:23/9 NXB XIC B9:22/10 XIO B3:0/1 BND OTE B9:22/10 NXB BST XIC B3:23/9 NXB XIC B9:22/11 XIO B3:0/1 XIO B3:0/0 BND OTE B9:22/11 BND EOR
%   B3:23/9  "TT-7050 LO TRIGGER BIT" %
%   B9:22/10  TT_7050_LO_ALM  "TT-7050 LO ALARM BIT" %
%   B3:0/1  ALARM_RESET  "ALARM RESET" %
%   B9:22/11  TT_7050_LO_ALT  "TT-7050 LO ALERT BIT" %
%   B3:0/0  ALARM_SILENCE  "ALARM SILENCE PUSHBUTTON" %
% Rung: 382 %
SOR GRT N11:91 0 GRT F8:45 F10:91 XIO B3:0/1 BST TON T4:91 1.0 0 0 NXB XIC T4:91/DN OSR B3:23/10 OTE B3:23/11 BND EOR
%   N11:91  TT_7050_HIALM_DLY_SP  "TT-7050 HI ALARM DELAY SP FROM HMI" %
%   F8:45  TT_7050_SCI  "TT-7050 SCALED INPUT" %
%   F10:91  TT_7050_HIALM_SP  "TT-7050 HI ALARM SP" %
%   B3:0/1  ALARM_RESET  "ALARM RESET" %
%   T4:91  TT_7050_HIALM_DLY_TM  "TT-7050 HI ALARM DELAY" %
%   B3:23/10  "OSR" %
%   B3:23/11  "TT-7050 HI TRIGGER BIT" %

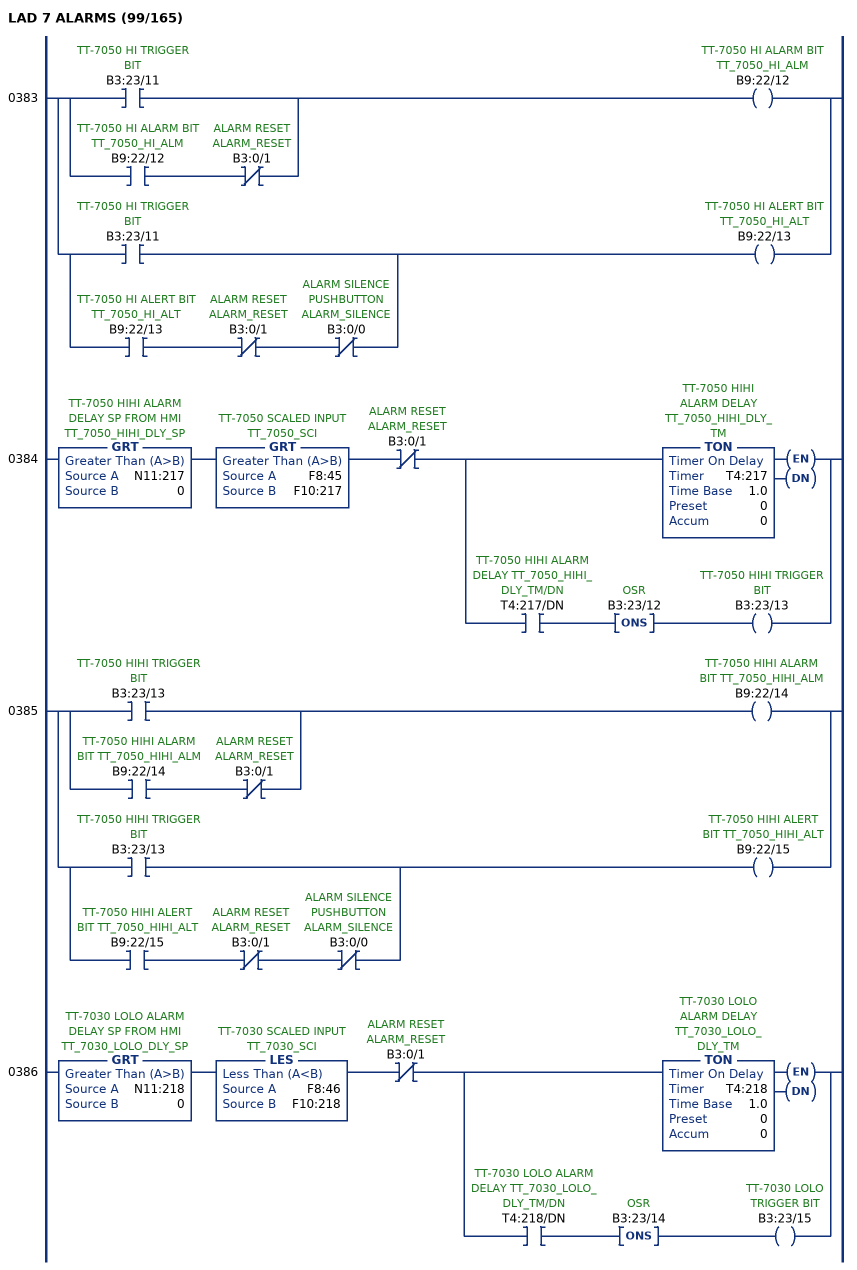
% Rung: 383 %
SOR BST BST XIC B3:23/11 NXB XIC B9:22/12 XIO B3:0/1 BND OTE B9:22/12 NXB BST XIC B3:23/11 NXB XIC B9:22/13 XIO B3:0/1 XIO B3:0/0 BND OTE B9:22/13 BND EOR
%   B3:23/11  "TT-7050 HI TRIGGER BIT" %
%   B9:22/12  TT_7050_HI_ALM  "TT-7050 HI ALARM BIT" %
%   B3:0/1  ALARM_RESET  "ALARM RESET" %
%   B9:22/13  TT_7050_HI_ALT  "TT-7050 HI ALERT BIT" %
%   B3:0/0  ALARM_SILENCE  "ALARM SILENCE PUSHBUTTON" %
% Rung: 384 %
SOR GRT N11:217 0 GRT F8:45 F10:217 XIO B3:0/1 BST TON T4:217 1.0 0 0 NXB XIC T4:217/DN OSR B3:23/12 OTE B3:23/13 BND EOR
%   N11:217  TT_7050_HIHI_DLY_SP  "TT-7050 HIHI ALARM DELAY SP FROM HMI" %
%   F8:45  TT_7050_SCI  "TT-7050 SCALED INPUT" %
%   F10:217  TT_7050_HIHI_SP  "TT-7050 HIHI ALARM SP" %
%   B3:0/1  ALARM_RESET  "ALARM RESET" %
%   T4:217  TT_7050_HIHI_DLY_TM  "TT-7050 HIHI ALARM DELAY" %
%   B3:23/12  "OSR" %
%   B3:23/13  "TT-7050 HIHI TRIGGER BIT" %
% Rung: 385 %
SOR BST BST XIC B3:23/13 NXB XIC B9:22/14 XIO B3:0/1 BND OTE B9:22/14 NXB BST XIC B3:23/13 NXB XIC B9:22/15 XIO B3:0/1 XIO B3:0/0 BND OTE B9:22/15 BND EOR
%   B3:23/13  "TT-7050 HIHI TRIGGER BIT" %
%   B9:22/14  TT_7050_HIHI_ALM  "TT-7050 HIHI ALARM BIT" %
%   B3:0/1  ALARM_RESET  "ALARM RESET" %
%   B9:22/15  TT_7050_HIHI_ALT  "TT-7050 HIHI ALERT BIT" %
%   B3:0/0  ALARM_SILENCE  "ALARM SILENCE PUSHBUTTON" %
% Rung: 386 %
SOR GRT N11:218 0 LES F8:46 F10:218 XIO B3:0/1 BST TON T4:218 1.0 0 0 NXB XIC T4:218/DN OSR B3:23/14 OTE B3:23/15 BND EOR
%   N11:218  TT_7030_LOLO_DLY_SP  "TT-7030 LOLO ALARM DELAY SP FROM HMI" %
%   F8:46  TT_7030_SCI  "TT-7030 SCALED INPUT" %
%   F10:218  TT_7030_LOLO_SP  "TT-7030 LOLO ALARM SP" %
%   B3:0/1  ALARM_RESET  "ALARM RESET" %
%   T4:218  TT_7030_LOLO_DLY_TM  "TT-7030 LOLO ALARM DELAY" %
%   B3:23/14  "OSR" %
%   B3:23/15  "TT-7030 LOLO TRIGGER BIT" %

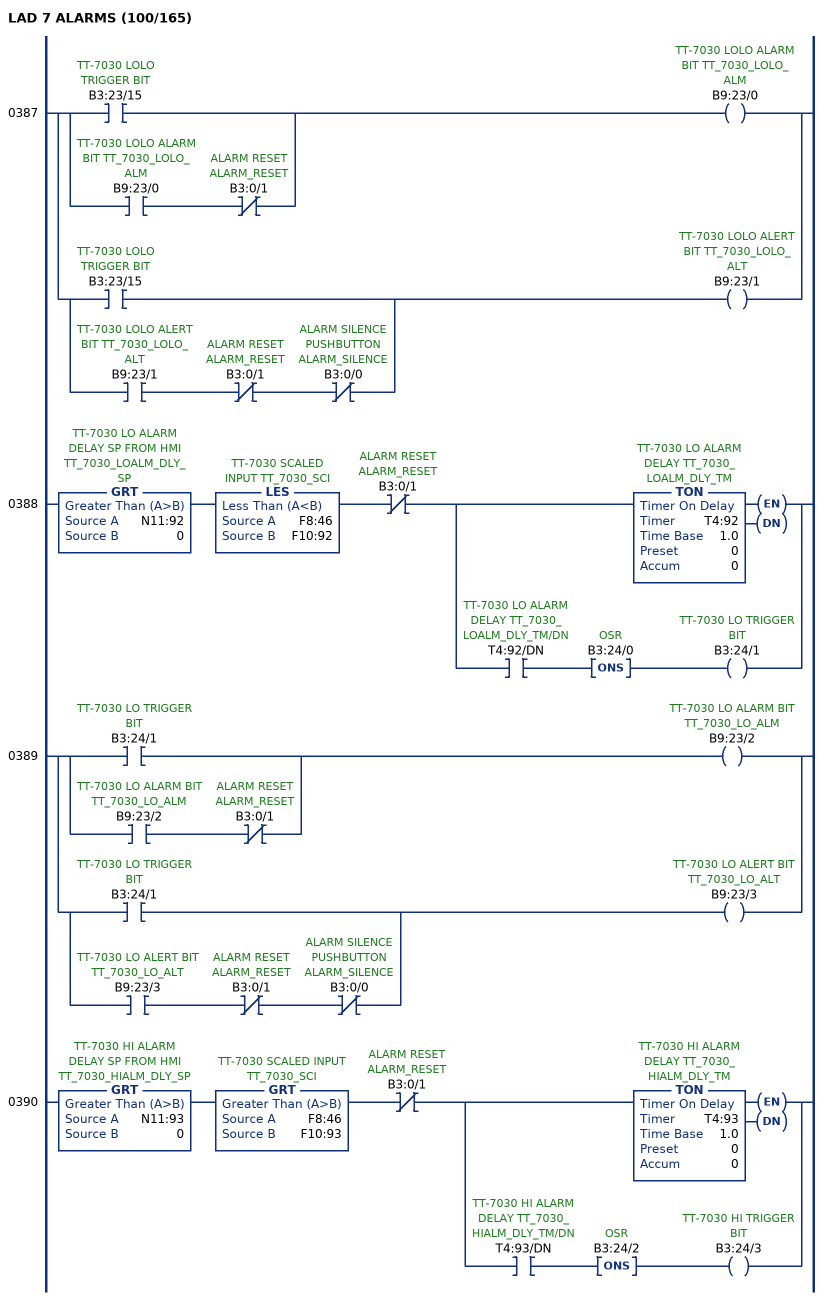
% Rung: 387 %
SOR BST BST XIC B3:23/15 NXB XIC B9:23/0 XIO B3:0/1 BND OTE B9:23/0 NXB BST XIC B3:23/15 NXB XIC B9:23/1 XIO B3:0/1 XIO B3:0/0 BND OTE B9:23/1 BND EOR
%   B3:23/15  "TT-7030 LOLO TRIGGER BIT" %
%   B9:23/0  TT_7030_LOLO_ALM  "TT-7030 LOLO ALARM BIT" %
%   B3:0/1  ALARM_RESET  "ALARM RESET" %
%   B9:23/1  TT_7030_LOLO_ALT  "TT-7030 LOLO ALERT BIT" %
%   B3:0/0  ALARM_SILENCE  "ALARM SILENCE PUSHBUTTON" %
% Rung: 388 %
SOR GRT N11:92 0 LES F8:46 F10:92 XIO B3:0/1 BST TON T4:92 1.0 0 0 NXB XIC T4:92/DN OSR B3:24/0 OTE B3:24/1 BND EOR
%   N11:92  TT_7030_LOALM_DLY_SP  "TT-7030 LO ALARM DELAY SP FROM HMI" %
%   F8:46  TT_7030_SCI  "TT-7030 SCALED INPUT" %
%   F10:92  TT_7030_LOALM_SP  "TT-7030 LO ALARM SP" %
%   B3:0/1  ALARM_RESET  "ALARM RESET" %
%   T4:92  TT_7030_LOALM_DLY_TM  "TT-7030 LO ALARM DELAY" %
%   B3:24/0  "OSR" %
%   B3:24/1  "TT-7030 LO TRIGGER BIT" %
% Rung: 389 %
SOR BST BST XIC B3:24/1 NXB XIC B9:23/2 XIO B3:0/1 BND OTE B9:23/2 NXB BST XIC B3:24/1 NXB XIC B9:23/3 XIO B3:0/1 XIO B3:0/0 BND OTE B9:23/3 BND EOR
%   B3:24/1  "TT-7030 LO TRIGGER BIT" %
%   B9:23/2  TT_7030_LO_ALM  "TT-7030 LO ALARM BIT" %
%   B3:0/1  ALARM_RESET  "ALARM RESET" %
%   B9:23/3  TT_7030_LO_ALT  "TT-7030 LO ALERT BIT" %
%   B3:0/0  ALARM_SILENCE  "ALARM SILENCE PUSHBUTTON" %
% Rung: 390 %
SOR GRT N11:93 0 GRT F8:46 F10:93 XIO B3:0/1 BST TON T4:93 1.0 0 0 NXB XIC T4:93/DN OSR B3:24/2 OTE B3:24/3 BND EOR
%   N11:93  TT_7030_HIALM_DLY_SP  "TT-7030 HI ALARM DELAY SP FROM HMI" %
%   F8:46  TT_7030_SCI  "TT-7030 SCALED INPUT" %
%   F10:93  TT_7030_HIALM_SP  "TT-7030 HI ALARM SP" %
%   B3:0/1  ALARM_RESET  "ALARM RESET" %
%   T4:93  TT_7030_HIALM_DLY_TM  "TT-7030 HI ALARM DELAY" %
%   B3:24/2  "OSR" %
%   B3:24/3  "TT-7030 HI TRIGGER BIT" %

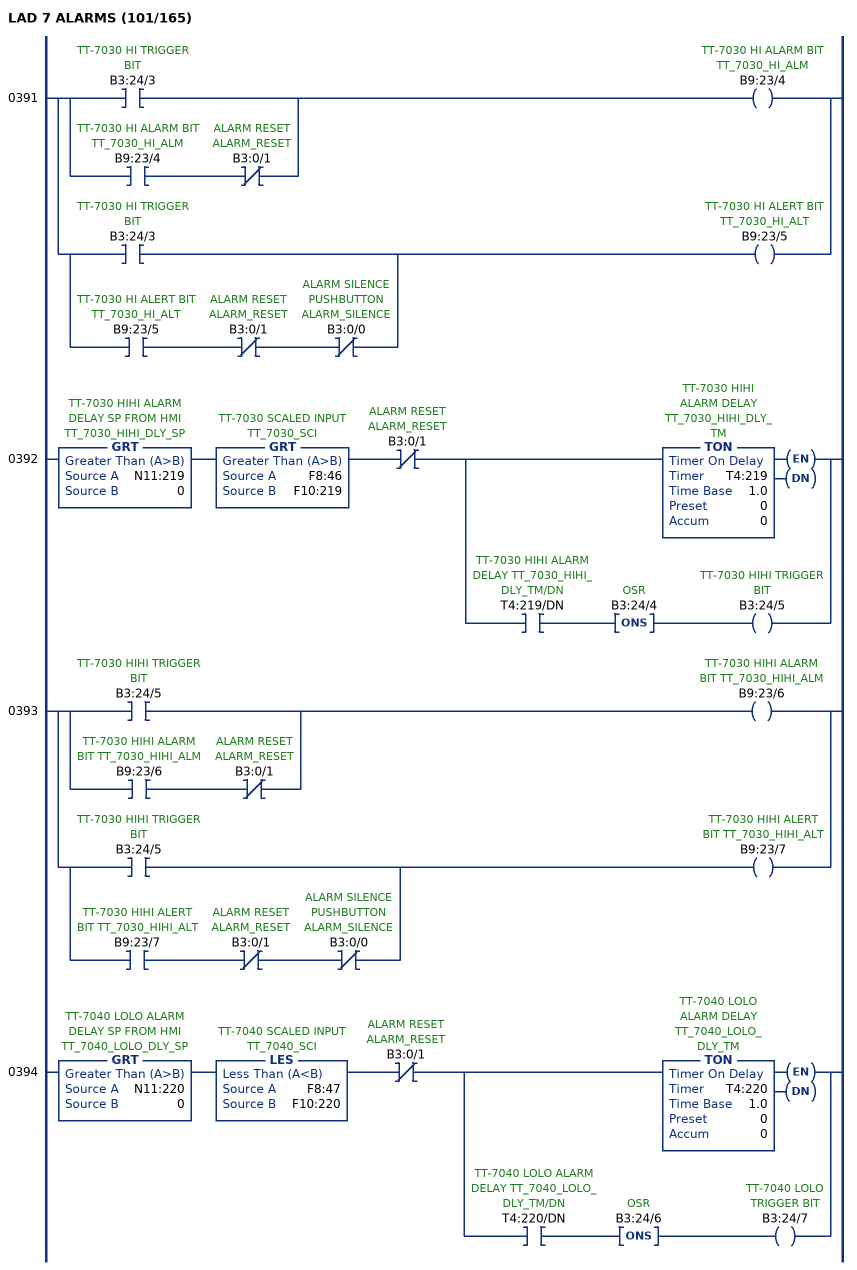
% Rung: 391 %
SOR BST BST XIC B3:24/3 NXB XIC B9:23/4 XIO B3:0/1 BND OTE B9:23/4 NXB BST XIC B3:24/3 NXB XIC B9:23/5 XIO B3:0/1 XIO B3:0/0 BND OTE B9:23/5 BND EOR
%   B3:24/3  "TT-7030 HI TRIGGER BIT" %
%   B9:23/4  TT_7030_HI_ALM  "TT-7030 HI ALARM BIT" %
%   B3:0/1  ALARM_RESET  "ALARM RESET" %
%   B9:23/5  TT_7030_HI_ALT  "TT-7030 HI ALERT BIT" %
%   B3:0/0  ALARM_SILENCE  "ALARM SILENCE PUSHBUTTON" %
% Rung: 392 %
SOR GRT N11:219 0 GRT F8:46 F10:219 XIO B3:0/1 BST TON T4:219 1.0 0 0 NXB XIC T4:219/DN OSR B3:24/4 OTE B3:24/5 BND EOR
%   N11:219  TT_7030_HIHI_DLY_SP  "TT-7030 HIHI ALARM DELAY SP FROM HMI" %
%   F8:46  TT_7030_SCI  "TT-7030 SCALED INPUT" %
%   F10:219  TT_7030_HIHI_SP  "TT-7030 HIHI ALARM SP" %
%   B3:0/1  ALARM_RESET  "ALARM RESET" %
%   T4:219  TT_7030_HIHI_DLY_TM  "TT-7030 HIHI ALARM DELAY" %
%   B3:24/4  "OSR" %
%   B3:24/5  "TT-7030 HIHI TRIGGER BIT" %
% Rung: 393 %
SOR BST BST XIC B3:24/5 NXB XIC B9:23/6 XIO B3:0/1 BND OTE B9:23/6 NXB BST XIC B3:24/5 NXB XIC B9:23/7 XIO B3:0/1 XIO B3:0/0 BND OTE B9:23/7 BND EOR
%   B3:24/5  "TT-7030 HIHI TRIGGER BIT" %
%   B9:23/6  TT_7030_HIHI_ALM  "TT-7030 HIHI ALARM BIT" %
%   B3:0/1  ALARM_RESET  "ALARM RESET" %
%   B9:23/7  TT_7030_HIHI_ALT  "TT-7030 HIHI ALERT BIT" %
%   B3:0/0  ALARM_SILENCE  "ALARM SILENCE PUSHBUTTON" %
% Rung: 394 %
SOR GRT N11:220 0 LES F8:47 F10:220 XIO B3:0/1 BST TON T4:220 1.0 0 0 NXB XIC T4:220/DN OSR B3:24/6 OTE B3:24/7 BND EOR
%   N11:220  TT_7040_LOLO_DLY_SP  "TT-7040 LOLO ALARM DELAY SP FROM HMI" %
%   F8:47  TT_7040_SCI  "TT-7040 SCALED INPUT" %
%   F10:220  TT_7040_LOLO_SP  "TT-7040 LOLO ALARM SP" %
%   B3:0/1  ALARM_RESET  "ALARM RESET" %
%   T4:220  TT_7040_LOLO_DLY_TM  "TT-7040 LOLO ALARM DELAY" %
%   B3:24/6  "OSR" %
%   B3:24/7  "TT-7040 LOLO TRIGGER BIT" %

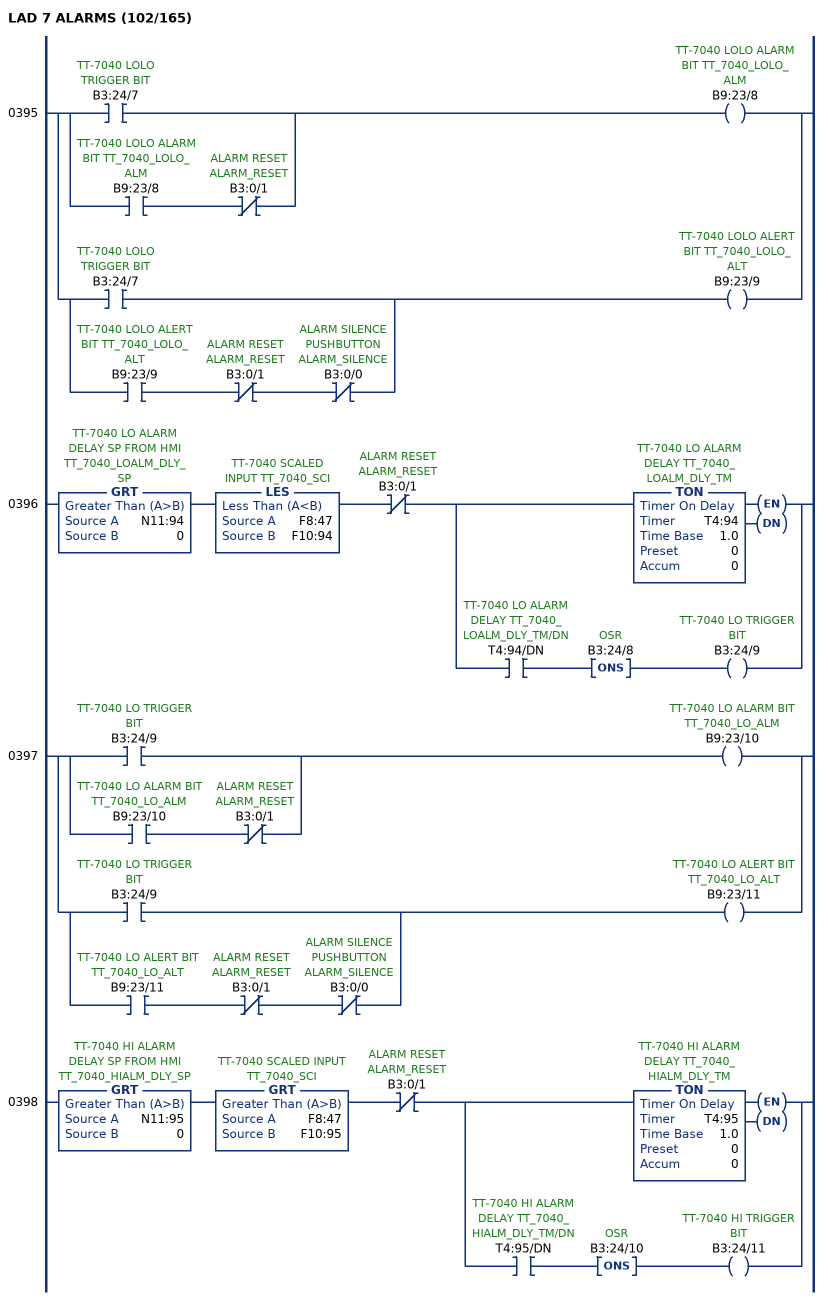
% Rung: 395 %
SOR BST BST XIC B3:24/7 NXB XIC B9:23/8 XIO B3:0/1 BND OTE B9:23/8 NXB BST XIC B3:24/7 NXB XIC B9:23/9 XIO B3:0/1 XIO B3:0/0 BND OTE B9:23/9 BND EOR
%   B3:24/7  "TT-7040 LOLO TRIGGER BIT" %
%   B9:23/8  TT_7040_LOLO_ALM  "TT-7040 LOLO ALARM BIT" %
%   B3:0/1  ALARM_RESET  "ALARM RESET" %
%   B9:23/9  TT_7040_LOLO_ALT  "TT-7040 LOLO ALERT BIT" %
%   B3:0/0  ALARM_SILENCE  "ALARM SILENCE PUSHBUTTON" %
% Rung: 396 %
SOR GRT N11:94 0 LES F8:47 F10:94 XIO B3:0/1 BST TON T4:94 1.0 0 0 NXB XIC T4:94/DN OSR B3:24/8 OTE B3:24/9 BND EOR
%   N11:94  TT_7040_LOALM_DLY_SP  "TT-7040 LO ALARM DELAY SP FROM HMI" %
%   F8:47  TT_7040_SCI  "TT-7040 SCALED INPUT" %
%   F10:94  TT_7040_LOALM_SP  "TT-7040 LO ALARM SP" %
%   B3:0/1  ALARM_RESET  "ALARM RESET" %
%   T4:94  TT_7040_LOALM_DLY_TM  "TT-7040 LO ALARM DELAY" %
%   B3:24/8  "OSR" %
%   B3:24/9  "TT-7040 LO TRIGGER BIT" %
% Rung: 397 %
SOR BST BST XIC B3:24/9 NXB XIC B9:23/10 XIO B3:0/1 BND OTE B9:23/10 NXB BST XIC B3:24/9 NXB XIC B9:23/11 XIO B3:0/1 XIO B3:0/0 BND OTE B9:23/11 BND EOR
%   B3:24/9  "TT-7040 LO TRIGGER BIT" %
%   B9:23/10  TT_7040_LO_ALM  "TT-7040 LO ALARM BIT" %
%   B3:0/1  ALARM_RESET  "ALARM RESET" %
%   B9:23/11  TT_7040_LO_ALT  "TT-7040 LO ALERT BIT" %
%   B3:0/0  ALARM_SILENCE  "ALARM SILENCE PUSHBUTTON" %
% Rung: 398 %
SOR GRT N11:95 0 GRT F8:47 F10:95 XIO B3:0/1 BST TON T4:95 1.0 0 0 NXB XIC T4:95/DN OSR B3:24/10 OTE B3:24/11 BND EOR
%   N11:95  TT_7040_HIALM_DLY_SP  "TT-7040 HI ALARM DELAY SP FROM HMI" %
%   F8:47  TT_7040_SCI  "TT-7040 SCALED INPUT" %
%   F10:95  TT_7040_HIALM_SP  "TT-7040 HI ALARM SP" %
%   B3:0/1  ALARM_RESET  "ALARM RESET" %
%   T4:95  TT_7040_HIALM_DLY_TM  "TT-7040 HI ALARM DELAY" %
%   B3:24/10  "OSR" %
%   B3:24/11  "TT-7040 HI TRIGGER BIT" %

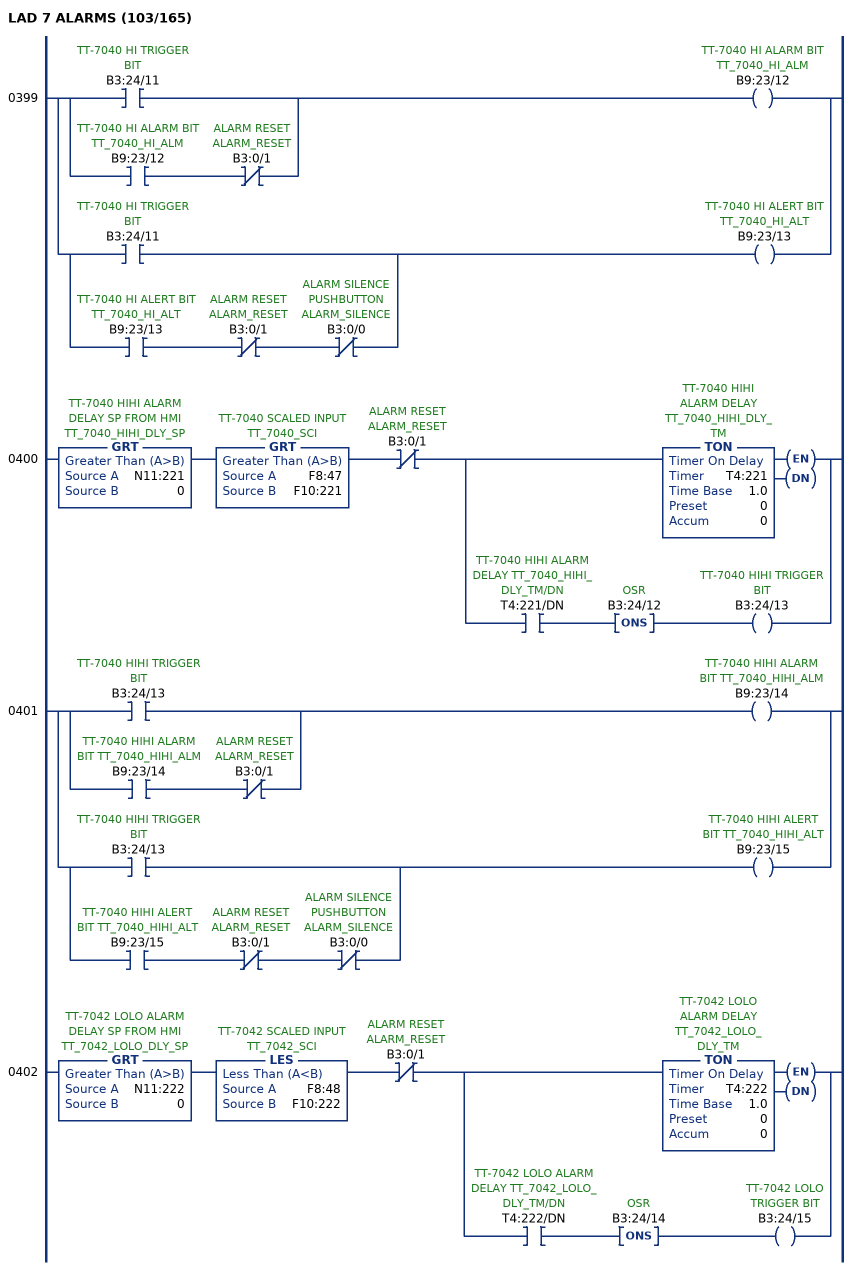
% Rung: 399 %
SOR BST BST XIC B3:24/11 NXB XIC B9:23/12 XIO B3:0/1 BND OTE B9:23/12 NXB BST XIC B3:24/11 NXB XIC B9:23/13 XIO B3:0/1 XIO B3:0/0 BND OTE B9:23/13 BND EOR
%   B3:24/11  "TT-7040 HI TRIGGER BIT" %
%   B9:23/12  TT_7040_HI_ALM  "TT-7040 HI ALARM BIT" %
%   B3:0/1  ALARM_RESET  "ALARM RESET" %
%   B9:23/13  TT_7040_HI_ALT  "TT-7040 HI ALERT BIT" %
%   B3:0/0  ALARM_SILENCE  "ALARM SILENCE PUSHBUTTON" %
% Rung: 400 %
SOR GRT N11:221 0 GRT F8:47 F10:221 XIO B3:0/1 BST TON T4:221 1.0 0 0 NXB XIC T4:221/DN OSR B3:24/12 OTE B3:24/13 BND EOR
%   N11:221  TT_7040_HIHI_DLY_SP  "TT-7040 HIHI ALARM DELAY SP FROM HMI" %
%   F8:47  TT_7040_SCI  "TT-7040 SCALED INPUT" %
%   F10:221  TT_7040_HIHI_SP  "TT-7040 HIHI ALARM SP" %
%   B3:0/1  ALARM_RESET  "ALARM RESET" %
%   T4:221  TT_7040_HIHI_DLY_TM  "TT-7040 HIHI ALARM DELAY" %
%   B3:24/12  "OSR" %
%   B3:24/13  "TT-7040 HIHI TRIGGER BIT" %
% Rung: 401 %
SOR BST BST XIC B3:24/13 NXB XIC B9:23/14 XIO B3:0/1 BND OTE B9:23/14 NXB BST XIC B3:24/13 NXB XIC B9:23/15 XIO B3:0/1 XIO B3:0/0 BND OTE B9:23/15 BND EOR
%   B3:24/13  "TT-7040 HIHI TRIGGER BIT" %
%   B9:23/14  TT_7040_HIHI_ALM  "TT-7040 HIHI ALARM BIT" %
%   B3:0/1  ALARM_RESET  "ALARM RESET" %
%   B9:23/15  TT_7040_HIHI_ALT  "TT-7040 HIHI ALERT BIT" %
%   B3:0/0  ALARM_SILENCE  "ALARM SILENCE PUSHBUTTON" %
% Rung: 402 %
SOR GRT N11:222 0 LES F8:48 F10:222 XIO B3:0/1 BST TON T4:222 1.0 0 0 NXB XIC T4:222/DN OSR B3:24/14 OTE B3:24/15 BND EOR
%   N11:222  TT_7042_LOLO_DLY_SP  "TT-7042 LOLO ALARM DELAY SP FROM HMI" %
%   F8:48  TT_7042_SCI  "TT-7042 SCALED INPUT" %
%   F10:222  TT_7042_LOLO_SP  "TT-7042 LOLO ALARM SP" %
%   B3:0/1  ALARM_RESET  "ALARM RESET" %
%   T4:222  TT_7042_LOLO_DLY_TM  "TT-7042 LOLO ALARM DELAY" %
%   B3:24/14  "OSR" %
%   B3:24/15  "TT-7042 LOLO TRIGGER BIT" %

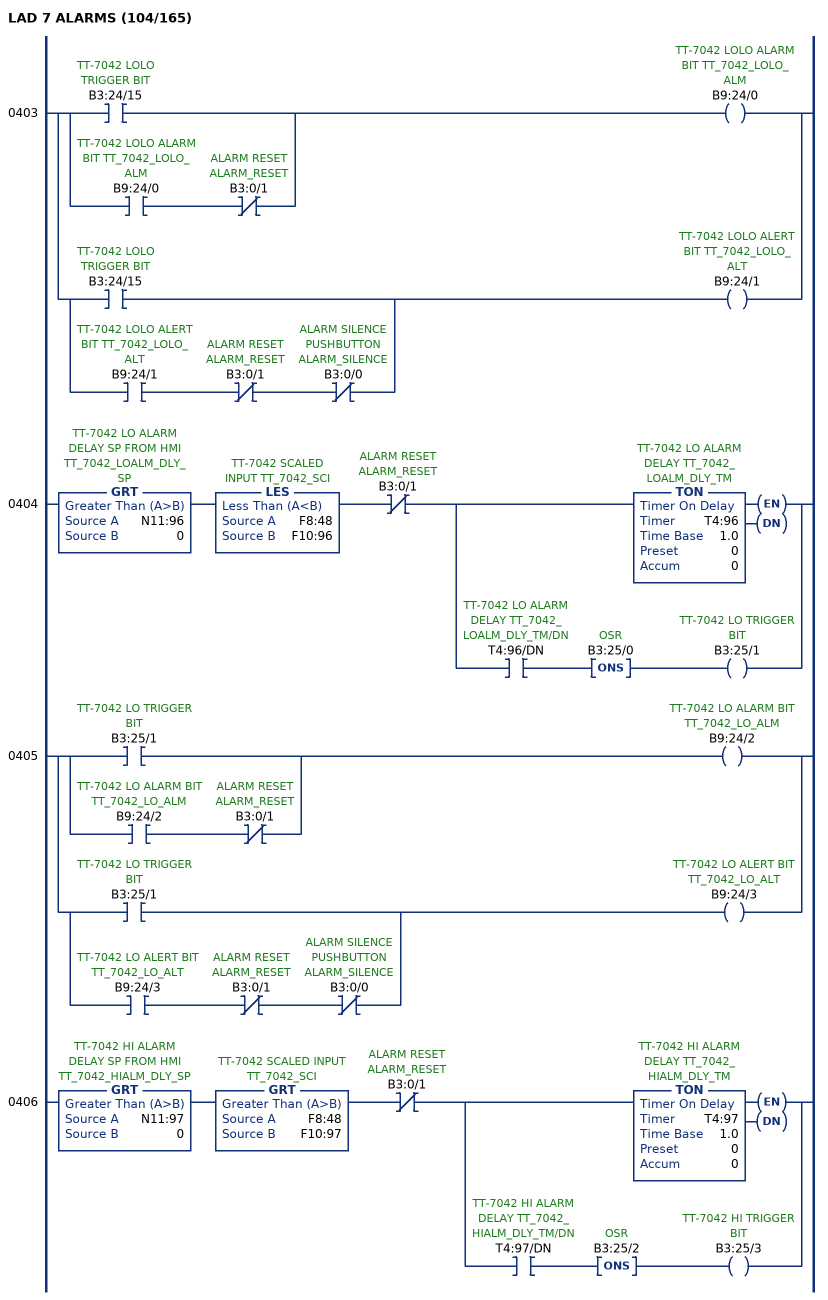
% Rung: 403 %
SOR BST BST XIC B3:24/15 NXB XIC B9:24/0 XIO B3:0/1 BND OTE B9:24/0 NXB BST XIC B3:24/15 NXB XIC B9:24/1 XIO B3:0/1 XIO B3:0/0 BND OTE B9:24/1 BND EOR
%   B3:24/15  "TT-7042 LOLO TRIGGER BIT" %
%   B9:24/0  TT_7042_LOLO_ALM  "TT-7042 LOLO ALARM BIT" %
%   B3:0/1  ALARM_RESET  "ALARM RESET" %
%   B9:24/1  TT_7042_LOLO_ALT  "TT-7042 LOLO ALERT BIT" %
%   B3:0/0  ALARM_SILENCE  "ALARM SILENCE PUSHBUTTON" %
% Rung: 404 %
SOR GRT N11:96 0 LES F8:48 F10:96 XIO B3:0/1 BST TON T4:96 1.0 0 0 NXB XIC T4:96/DN OSR B3:25/0 OTE B3:25/1 BND EOR
%   N11:96  TT_7042_LOALM_DLY_SP  "TT-7042 LO ALARM DELAY SP FROM HMI" %
%   F8:48  TT_7042_SCI  "TT-7042 SCALED INPUT" %
%   F10:96  TT_7042_LOALM_SP  "TT-7042 LO ALARM SP" %
%   B3:0/1  ALARM_RESET  "ALARM RESET" %
%   T4:96  TT_7042_LOALM_DLY_TM  "TT-7042 LO ALARM DELAY" %
%   B3:25/0  "OSR" %
%   B3:25/1  "TT-7042 LO TRIGGER BIT" %
% Rung: 405 %
SOR BST BST XIC B3:25/1 NXB XIC B9:24/2 XIO B3:0/1 BND OTE B9:24/2 NXB BST XIC B3:25/1 NXB XIC B9:24/3 XIO B3:0/1 XIO B3:0/0 BND OTE B9:24/3 BND EOR
%   B3:25/1  "TT-7042 LO TRIGGER BIT" %
%   B9:24/2  TT_7042_LO_ALM  "TT-7042 LO ALARM BIT" %
%   B3:0/1  ALARM_RESET  "ALARM RESET" %
%   B9:24/3  TT_7042_LO_ALT  "TT-7042 LO ALERT BIT" %
%   B3:0/0  ALARM_SILENCE  "ALARM SILENCE PUSHBUTTON" %
% Rung: 406 %
SOR GRT N11:97 0 GRT F8:48 F10:97 XIO B3:0/1 BST TON T4:97 1.0 0 0 NXB XIC T4:97/DN OSR B3:25/2 OTE B3:25/3 BND EOR
%   N11:97  TT_7042_HIALM_DLY_SP  "TT-7042 HI ALARM DELAY SP FROM HMI" %
%   F8:48  TT_7042_SCI  "TT-7042 SCALED INPUT" %
%   F10:97  TT_7042_HIALM_SP  "TT-7042 HI ALARM SP" %
%   B3:0/1  ALARM_RESET  "ALARM RESET" %
%   T4:97  TT_7042_HIALM_DLY_TM  "TT-7042 HI ALARM DELAY" %
%   B3:25/2  "OSR" %
%   B3:25/3  "TT-7042 HI TRIGGER BIT" %

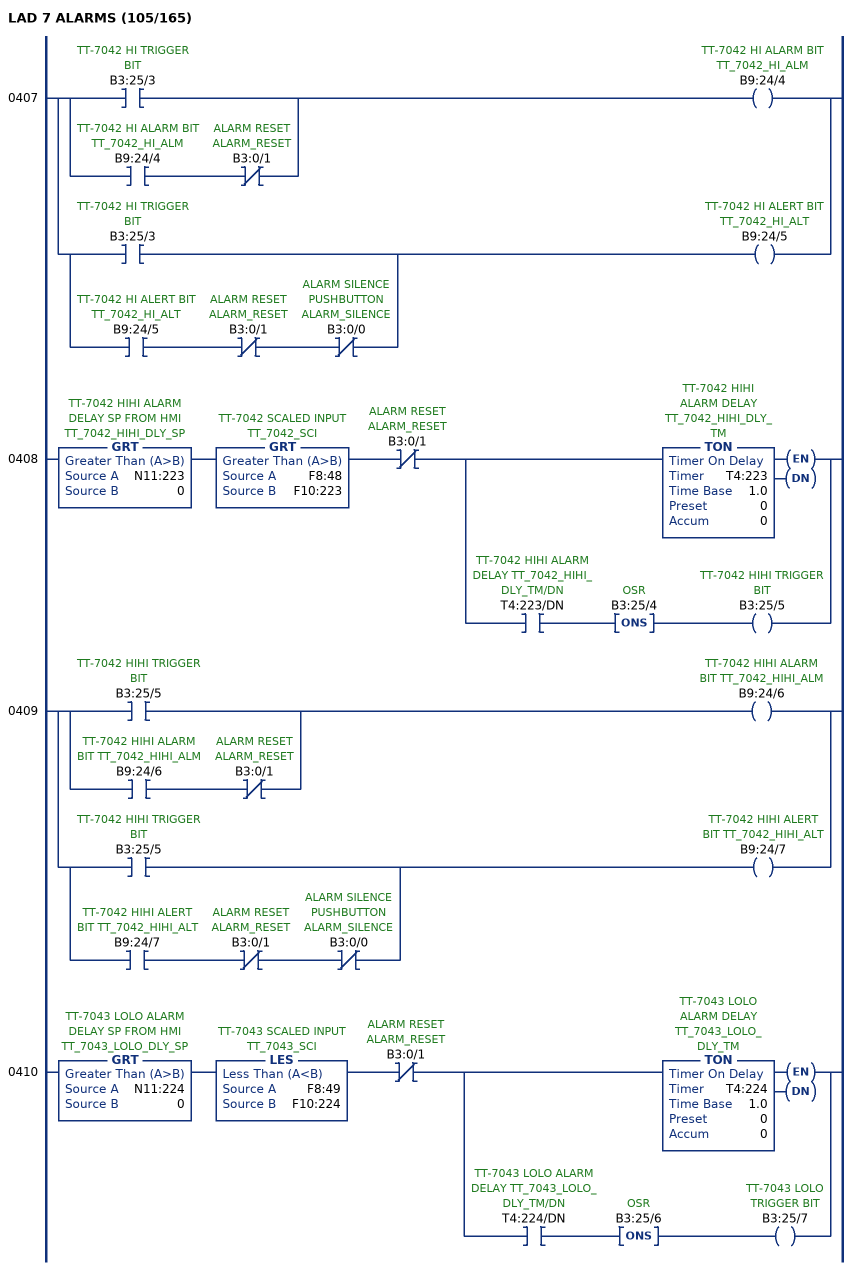
% Rung: 407 %
SOR BST BST XIC B3:25/3 NXB XIC B9:24/4 XIO B3:0/1 BND OTE B9:24/4 NXB BST XIC B3:25/3 NXB XIC B9:24/5 XIO B3:0/1 XIO B3:0/0 BND OTE B9:24/5 BND EOR
%   B3:25/3  "TT-7042 HI TRIGGER BIT" %
%   B9:24/4  TT_7042_HI_ALM  "TT-7042 HI ALARM BIT" %
%   B3:0/1  ALARM_RESET  "ALARM RESET" %
%   B9:24/5  TT_7042_HI_ALT  "TT-7042 HI ALERT BIT" %
%   B3:0/0  ALARM_SILENCE  "ALARM SILENCE PUSHBUTTON" %
% Rung: 408 %
SOR GRT N11:223 0 GRT F8:48 F10:223 XIO B3:0/1 BST TON T4:223 1.0 0 0 NXB XIC T4:223/DN OSR B3:25/4 OTE B3:25/5 BND EOR
%   N11:223  TT_7042_HIHI_DLY_SP  "TT-7042 HIHI ALARM DELAY SP FROM HMI" %
%   F8:48  TT_7042_SCI  "TT-7042 SCALED INPUT" %
%   F10:223  TT_7042_HIHI_SP  "TT-7042 HIHI ALARM SP" %
%   B3:0/1  ALARM_RESET  "ALARM RESET" %
%   T4:223  TT_7042_HIHI_DLY_TM  "TT-7042 HIHI ALARM DELAY" %
%   B3:25/4  "OSR" %
%   B3:25/5  "TT-7042 HIHI TRIGGER BIT" %
% Rung: 409 %
SOR BST BST XIC B3:25/5 NXB XIC B9:24/6 XIO B3:0/1 BND OTE B9:24/6 NXB BST XIC B3:25/5 NXB XIC B9:24/7 XIO B3:0/1 XIO B3:0/0 BND OTE B9:24/7 BND EOR
%   B3:25/5  "TT-7042 HIHI TRIGGER BIT" %
%   B9:24/6  TT_7042_HIHI_ALM  "TT-7042 HIHI ALARM BIT" %
%   B3:0/1  ALARM_RESET  "ALARM RESET" %
%   B9:24/7  TT_7042_HIHI_ALT  "TT-7042 HIHI ALERT BIT" %
%   B3:0/0  ALARM_SILENCE  "ALARM SILENCE PUSHBUTTON" %
% Rung: 410 %
SOR GRT N11:224 0 LES F8:49 F10:224 XIO B3:0/1 BST TON T4:224 1.0 0 0 NXB XIC T4:224/DN OSR B3:25/6 OTE B3:25/7 BND EOR
%   N11:224  TT_7043_LOLO_DLY_SP  "TT-7043 LOLO ALARM DELAY SP FROM HMI" %
%   F8:49  TT_7043_SCI  "TT-7043 SCALED INPUT" %
%   F10:224  TT_7043_LOLO_SP  "TT-7043L LOLO ALARM SP" %
%   B3:0/1  ALARM_RESET  "ALARM RESET" %
%   T4:224  TT_7043_LOLO_DLY_TM  "TT-7043 LOLO ALARM DELAY" %
%   B3:25/6  "OSR" %
%   B3:25/7  "TT-7043 LOLO TRIGGER BIT" %

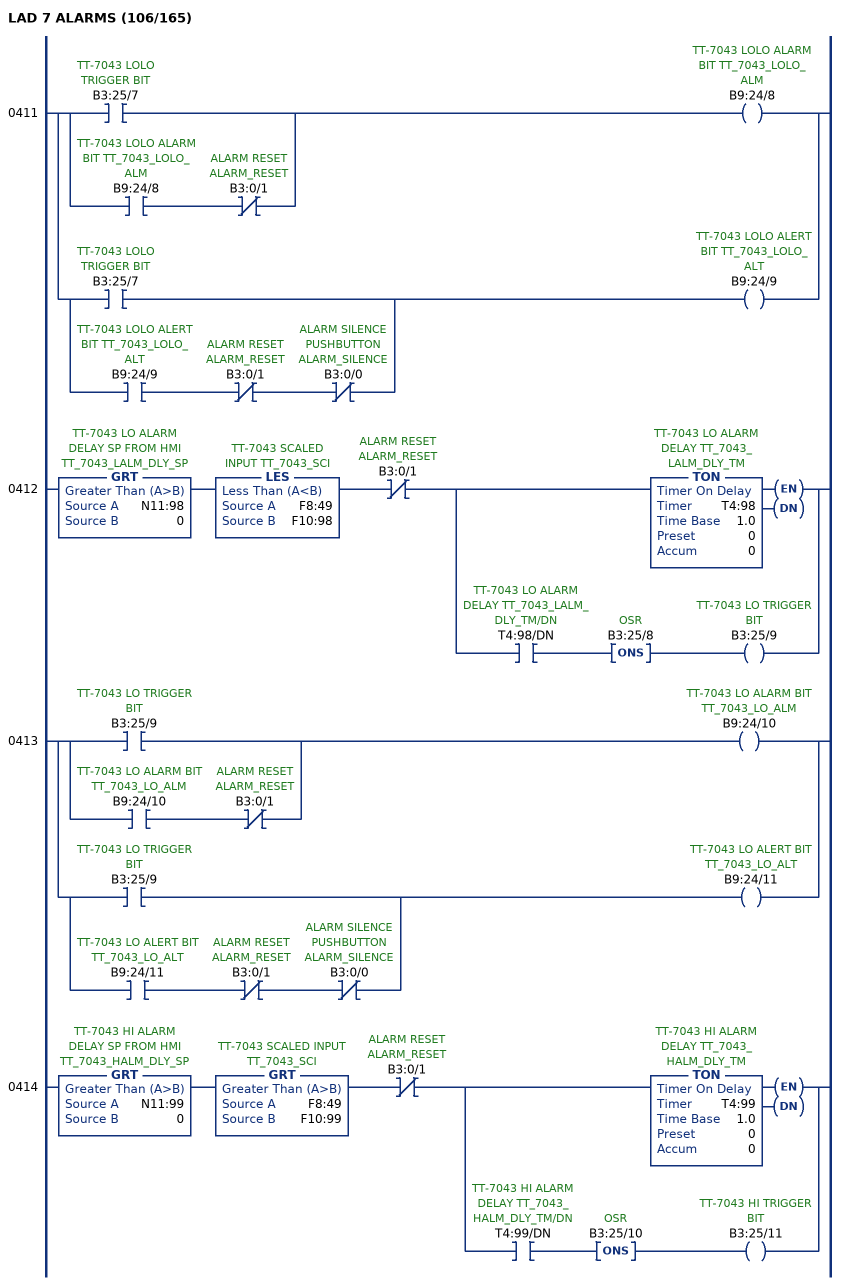
% Rung: 411 %
SOR BST BST XIC B3:25/7 NXB XIC B9:24/8 XIO B3:0/1 BND OTE B9:24/8 NXB BST XIC B3:25/7 NXB XIC B9:24/9 XIO B3:0/1 XIO B3:0/0 BND OTE B9:24/9 BND EOR
%   B3:25/7  "TT-7043 LOLO TRIGGER BIT" %
%   B9:24/8  TT_7043_LOLO_ALM  "TT-7043 LOLO ALARM BIT" %
%   B3:0/1  ALARM_RESET  "ALARM RESET" %
%   B9:24/9  TT_7043_LOLO_ALT  "TT-7043 LOLO ALERT BIT" %
%   B3:0/0  ALARM_SILENCE  "ALARM SILENCE PUSHBUTTON" %
% Rung: 412 %
SOR GRT N11:98 0 LES F8:49 F10:98 XIO B3:0/1 BST TON T4:98 1.0 0 0 NXB XIC T4:98/DN OSR B3:25/8 OTE B3:25/9 BND EOR
%   N11:98  TT_7043_LALM_DLY_SP  "TT-7043 LO ALARM DELAY SP FROM HMI" %
%   F8:49  TT_7043_SCI  "TT-7043 SCALED INPUT" %
%   F10:98  TT_7043_LOALM_SP  "TT-7043L LO ALARM SP" %
%   B3:0/1  ALARM_RESET  "ALARM RESET" %
%   T4:98  TT_7043_LALM_DLY_TM  "TT-7043 LO ALARM DELAY" %
%   B3:25/8  "OSR" %
%   B3:25/9  "TT-7043 LO TRIGGER BIT" %
% Rung: 413 %
SOR BST BST XIC B3:25/9 NXB XIC B9:24/10 XIO B3:0/1 BND OTE B9:24/10 NXB BST XIC B3:25/9 NXB XIC B9:24/11 XIO B3:0/1 XIO B3:0/0 BND OTE B9:24/11 BND EOR
%   B3:25/9  "TT-7043 LO TRIGGER BIT" %
%   B9:24/10  TT_7043_LO_ALM  "TT-7043 LO ALARM BIT" %
%   B3:0/1  ALARM_RESET  "ALARM RESET" %
%   B9:24/11  TT_7043_LO_ALT  "TT-7043 LO ALERT BIT" %
%   B3:0/0  ALARM_SILENCE  "ALARM SILENCE PUSHBUTTON" %
% Rung: 414 %
SOR GRT N11:99 0 GRT F8:49 F10:99 XIO B3:0/1 BST TON T4:99 1.0 0 0 NXB XIC T4:99/DN OSR B3:25/10 OTE B3:25/11 BND EOR
%   N11:99  TT_7043_HALM_DLY_SP  "TT-7043 HI ALARM DELAY SP FROM HMI" %
%   F8:49  TT_7043_SCI  "TT-7043 SCALED INPUT" %
%   F10:99  TT_7043_HIALM_SP  "TT-7043L HI ALARM SP" %
%   B3:0/1  ALARM_RESET  "ALARM RESET" %
%   T4:99  TT_7043_HALM_DLY_TM  "TT-7043 HI ALARM DELAY" %
%   B3:25/10  "OSR" %
%   B3:25/11  "TT-7043 HI TRIGGER BIT" %

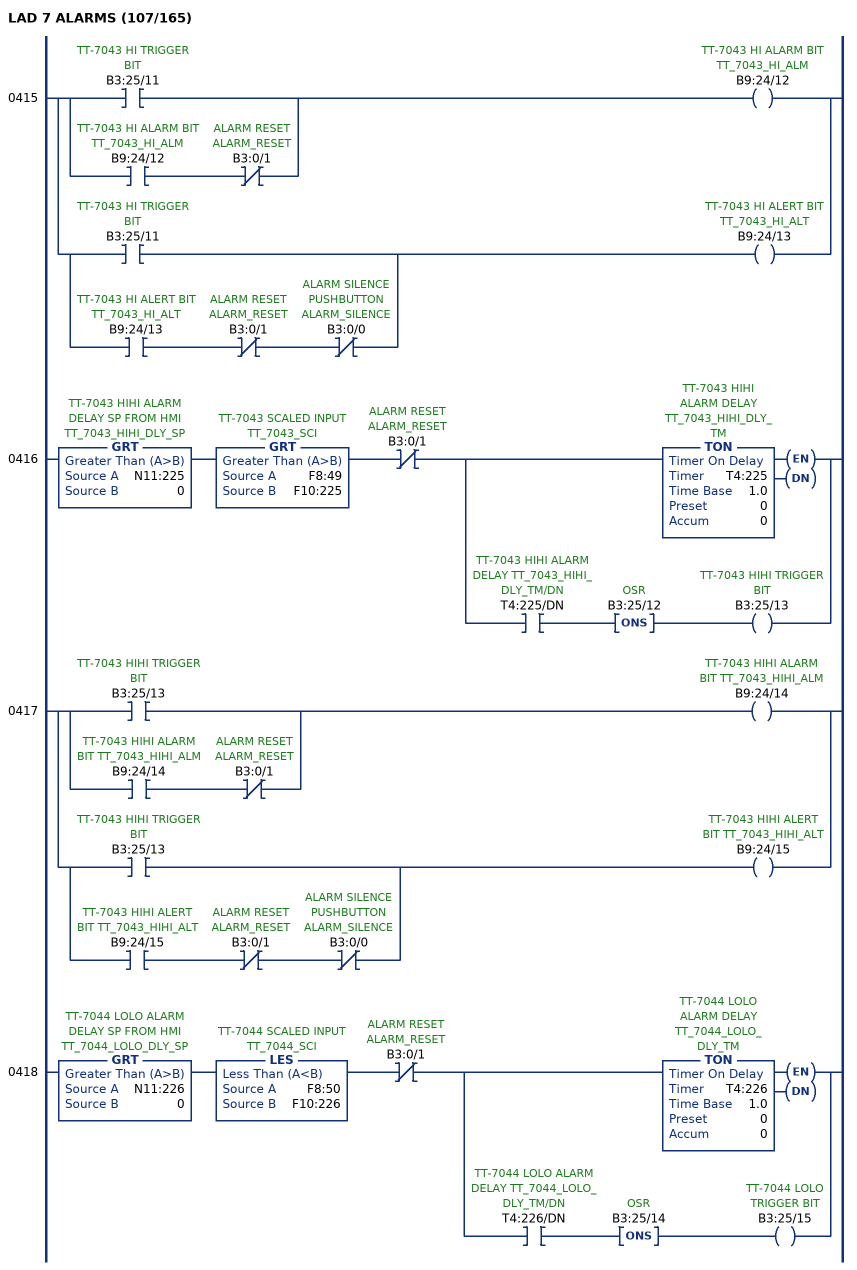
% Rung: 415 %
SOR BST BST XIC B3:25/11 NXB XIC B9:24/12 XIO B3:0/1 BND OTE B9:24/12 NXB BST XIC B3:25/11 NXB XIC B9:24/13 XIO B3:0/1 XIO B3:0/0 BND OTE B9:24/13 BND EOR
%   B3:25/11  "TT-7043 HI TRIGGER BIT" %
%   B9:24/12  TT_7043_HI_ALM  "TT-7043 HI ALARM BIT" %
%   B3:0/1  ALARM_RESET  "ALARM RESET" %
%   B9:24/13  TT_7043_HI_ALT  "TT-7043 HI ALERT BIT" %
%   B3:0/0  ALARM_SILENCE  "ALARM SILENCE PUSHBUTTON" %
% Rung: 416 %
SOR GRT N11:225 0 GRT F8:49 F10:225 XIO B3:0/1 BST TON T4:225 1.0 0 0 NXB XIC T4:225/DN OSR B3:25/12 OTE B3:25/13 BND EOR
%   N11:225  TT_7043_HIHI_DLY_SP  "TT-7043 HIHI ALARM DELAY SP FROM HMI" %
%   F8:49  TT_7043_SCI  "TT-7043 SCALED INPUT" %
%   F10:225  TT_7043_HIHI_SP  "TT-7043L HIHI ALARM SP" %
%   B3:0/1  ALARM_RESET  "ALARM RESET" %
%   T4:225  TT_7043_HIHI_DLY_TM  "TT-7043 HIHI ALARM DELAY" %
%   B3:25/12  "OSR" %
%   B3:25/13  "TT-7043 HIHI TRIGGER BIT" %
% Rung: 417 %
SOR BST BST XIC B3:25/13 NXB XIC B9:24/14 XIO B3:0/1 BND OTE B9:24/14 NXB BST XIC B3:25/13 NXB XIC B9:24/15 XIO B3:0/1 XIO B3:0/0 BND OTE B9:24/15 BND EOR
%   B3:25/13  "TT-7043 HIHI TRIGGER BIT" %
%   B9:24/14  TT_7043_HIHI_ALM  "TT-7043 HIHI ALARM BIT" %
%   B3:0/1  ALARM_RESET  "ALARM RESET" %
%   B9:24/15  TT_7043_HIHI_ALT  "TT-7043 HIHI ALERT BIT" %
%   B3:0/0  ALARM_SILENCE  "ALARM SILENCE PUSHBUTTON" %
% Rung: 418 %
SOR GRT N11:226 0 LES F8:50 F10:226 XIO B3:0/1 BST TON T4:226 1.0 0 0 NXB XIC T4:226/DN OSR B3:25/14 OTE B3:25/15 BND EOR
%   N11:226  TT_7044_LOLO_DLY_SP  "TT-7044 LOLO ALARM DELAY SP FROM HMI" %
%   F8:50  TT_7044_SCI  "TT-7044 SCALED INPUT" %
%   F10:226  TT_7044_LOLO_SP  "TT-7043R LOLO ALARM SP" %
%   B3:0/1  ALARM_RESET  "ALARM RESET" %
%   T4:226  TT_7044_LOLO_DLY_TM  "TT-7044 LOLO ALARM DELAY" %
%   B3:25/14  "OSR" %
%   B3:25/15  "TT-7044 LOLO TRIGGER BIT" %

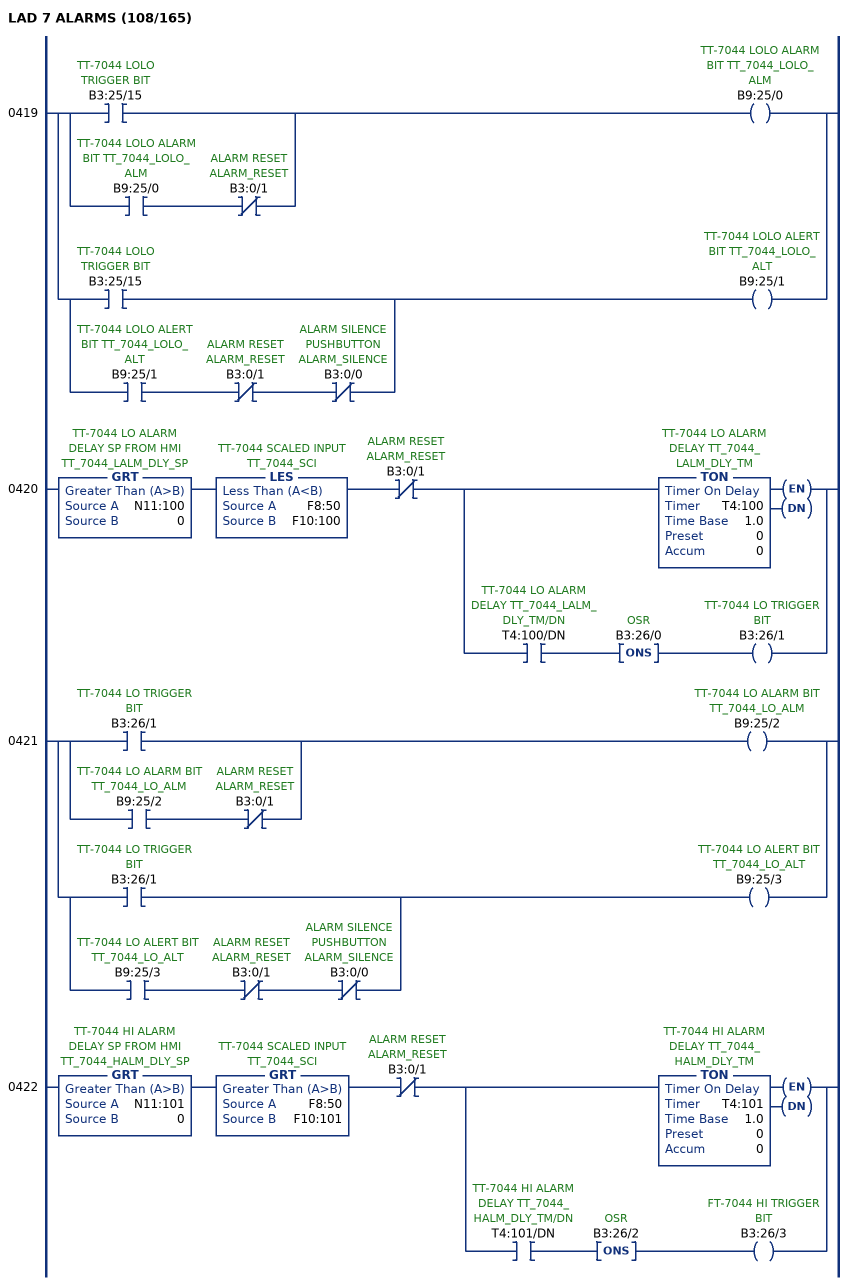
% Rung: 419 %
SOR BST BST XIC B3:25/15 NXB XIC B9:25/0 XIO B3:0/1 BND OTE B9:25/0 NXB BST XIC B3:25/15 NXB XIC B9:25/1 XIO B3:0/1 XIO B3:0/0 BND OTE B9:25/1 BND EOR
%   B3:25/15  "TT-7044 LOLO TRIGGER BIT" %
%   B9:25/0  TT_7044_LOLO_ALM  "TT-7044 LOLO ALARM BIT" %
%   B3:0/1  ALARM_RESET  "ALARM RESET" %
%   B9:25/1  TT_7044_LOLO_ALT  "TT-7044 LOLO ALERT BIT" %
%   B3:0/0  ALARM_SILENCE  "ALARM SILENCE PUSHBUTTON" %
% Rung: 420 %
SOR GRT N11:100 0 LES F8:50 F10:100 XIO B3:0/1 BST TON T4:100 1.0 0 0 NXB XIC T4:100/DN OSR B3:26/0 OTE B3:26/1 BND EOR
%   N11:100  TT_7044_LALM_DLY_SP  "TT-7044 LO ALARM DELAY SP FROM HMI" %
%   F8:50  TT_7044_SCI  "TT-7044 SCALED INPUT" %
%   F10:100  TT_7044_LOALM_SP  "TT-7043R LO ALARM SP" %
%   B3:0/1  ALARM_RESET  "ALARM RESET" %
%   T4:100  TT_7044_LALM_DLY_TM  "TT-7044 LO ALARM DELAY" %
%   B3:26/0  "OSR" %
%   B3:26/1  "TT-7044 LO TRIGGER BIT" %
% Rung: 421 %
SOR BST BST XIC B3:26/1 NXB XIC B9:25/2 XIO B3:0/1 BND OTE B9:25/2 NXB BST XIC B3:26/1 NXB XIC B9:25/3 XIO B3:0/1 XIO B3:0/0 BND OTE B9:25/3 BND EOR
%   B3:26/1  "TT-7044 LO TRIGGER BIT" %
%   B9:25/2  TT_7044_LO_ALM  "TT-7044 LO ALARM BIT" %
%   B3:0/1  ALARM_RESET  "ALARM RESET" %
%   B9:25/3  TT_7044_LO_ALT  "TT-7044 LO ALERT BIT" %
%   B3:0/0  ALARM_SILENCE  "ALARM SILENCE PUSHBUTTON" %
% Rung: 422 %
SOR GRT N11:101 0 GRT F8:50 F10:101 XIO B3:0/1 BST TON T4:101 1.0 0 0 NXB XIC T4:101/DN OSR B3:26/2 OTE B3:26/3 BND EOR
%   N11:101  TT_7044_HALM_DLY_SP  "TT-7044 HI ALARM DELAY SP FROM HMI" %
%   F8:50  TT_7044_SCI  "TT-7044 SCALED INPUT" %
%   F10:101  TT_7044_HIALM_SP  "TT-7043R HI ALARM SP" %
%   B3:0/1  ALARM_RESET  "ALARM RESET" %
%   T4:101  TT_7044_HALM_DLY_TM  "TT-7044 HI ALARM DELAY" %
%   B3:26/2  "OSR" %
%   B3:26/3  "FT-7044 HI TRIGGER BIT" %

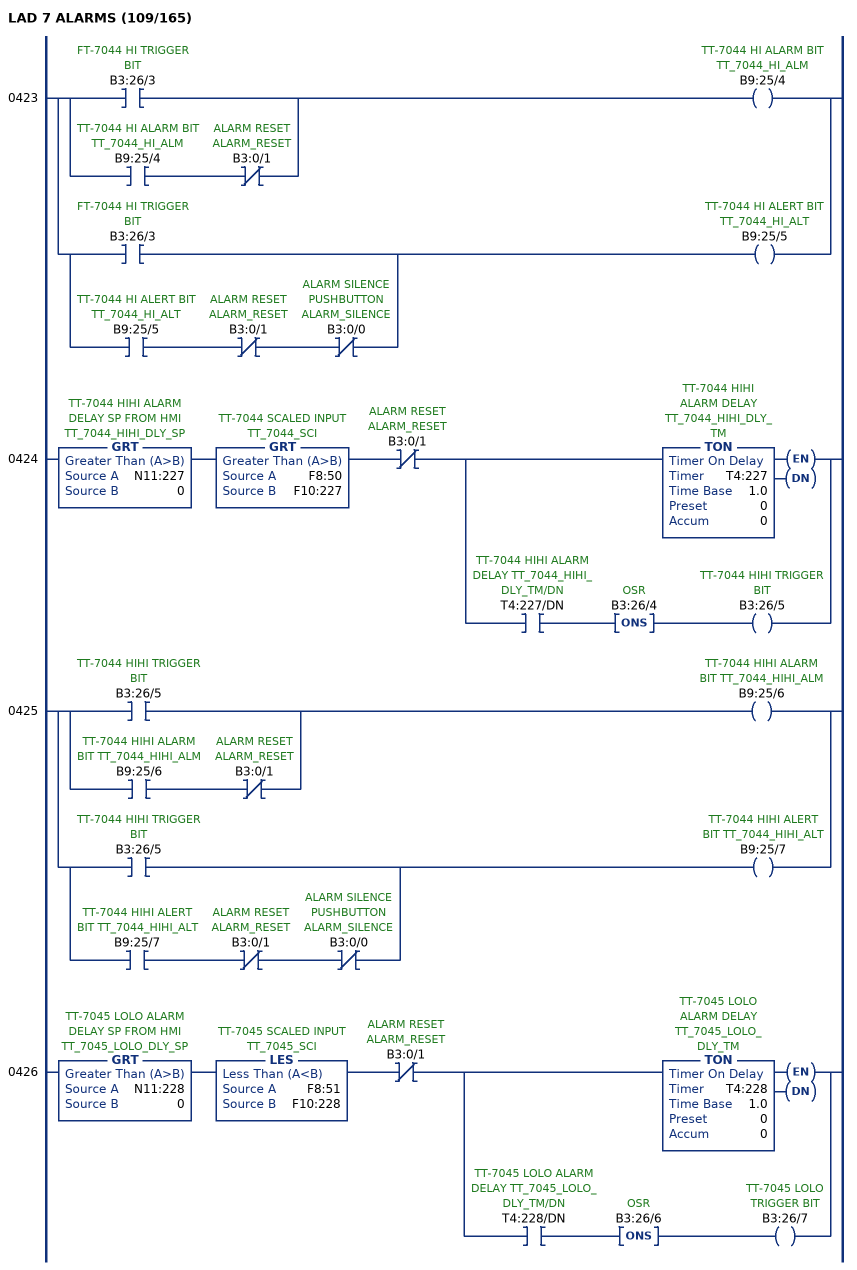
% Rung: 423 %
SOR BST BST XIC B3:26/3 NXB XIC B9:25/4 XIO B3:0/1 BND OTE B9:25/4 NXB BST XIC B3:26/3 NXB XIC B9:25/5 XIO B3:0/1 XIO B3:0/0 BND OTE B9:25/5 BND EOR
%   B3:26/3  "FT-7044 HI TRIGGER BIT" %
%   B9:25/4  TT_7044_HI_ALM  "TT-7044 HI ALARM BIT" %
%   B3:0/1  ALARM_RESET  "ALARM RESET" %
%   B9:25/5  TT_7044_HI_ALT  "TT-7044 HI ALERT BIT" %
%   B3:0/0  ALARM_SILENCE  "ALARM SILENCE PUSHBUTTON" %
% Rung: 424 %
SOR GRT N11:227 0 GRT F8:50 F10:227 XIO B3:0/1 BST TON T4:227 1.0 0 0 NXB XIC T4:227/DN OSR B3:26/4 OTE B3:26/5 BND EOR
%   N11:227  TT_7044_HIHI_DLY_SP  "TT-7044 HIHI ALARM DELAY SP FROM HMI" %
%   F8:50  TT_7044_SCI  "TT-7044 SCALED INPUT" %
%   F10:227  TT_7044_HIHI_SP  "TT-7043R HIHI ALARM SP" %
%   B3:0/1  ALARM_RESET  "ALARM RESET" %
%   T4:227  TT_7044_HIHI_DLY_TM  "TT-7044 HIHI ALARM DELAY" %
%   B3:26/4  "OSR" %
%   B3:26/5  "TT-7044 HIHI TRIGGER BIT" %
% Rung: 425 %
SOR BST BST XIC B3:26/5 NXB XIC B9:25/6 XIO B3:0/1 BND OTE B9:25/6 NXB BST XIC B3:26/5 NXB XIC B9:25/7 XIO B3:0/1 XIO B3:0/0 BND OTE B9:25/7 BND EOR
%   B3:26/5  "TT-7044 HIHI TRIGGER BIT" %
%   B9:25/6  TT_7044_HIHI_ALM  "TT-7044 HIHI ALARM BIT" %
%   B3:0/1  ALARM_RESET  "ALARM RESET" %
%   B9:25/7  TT_7044_HIHI_ALT  "TT-7044 HIHI ALERT BIT" %
%   B3:0/0  ALARM_SILENCE  "ALARM SILENCE PUSHBUTTON" %
% Rung: 426 %
SOR GRT N11:228 0 LES F8:51 F10:228 XIO B3:0/1 BST TON T4:228 1.0 0 0 NXB XIC T4:228/DN OSR B3:26/6 OTE B3:26/7 BND EOR
%   N11:228  TT_7045_LOLO_DLY_SP  "TT-7045 LOLO ALARM DELAY SP FROM HMI" %
%   F8:51  TT_7045_SCI  "TT-7045 SCALED INPUT" %
%   F10:228  TT_7045_LOLO_SP  "TT-7045 LOLO ALARM SP" %
%   B3:0/1  ALARM_RESET  "ALARM RESET" %
%   T4:228  TT_7045_LOLO_DLY_TM  "TT-7045 LOLO ALARM DELAY" %
%   B3:26/6  "OSR" %
%   B3:26/7  "TT-7045 LOLO TRIGGER BIT" %

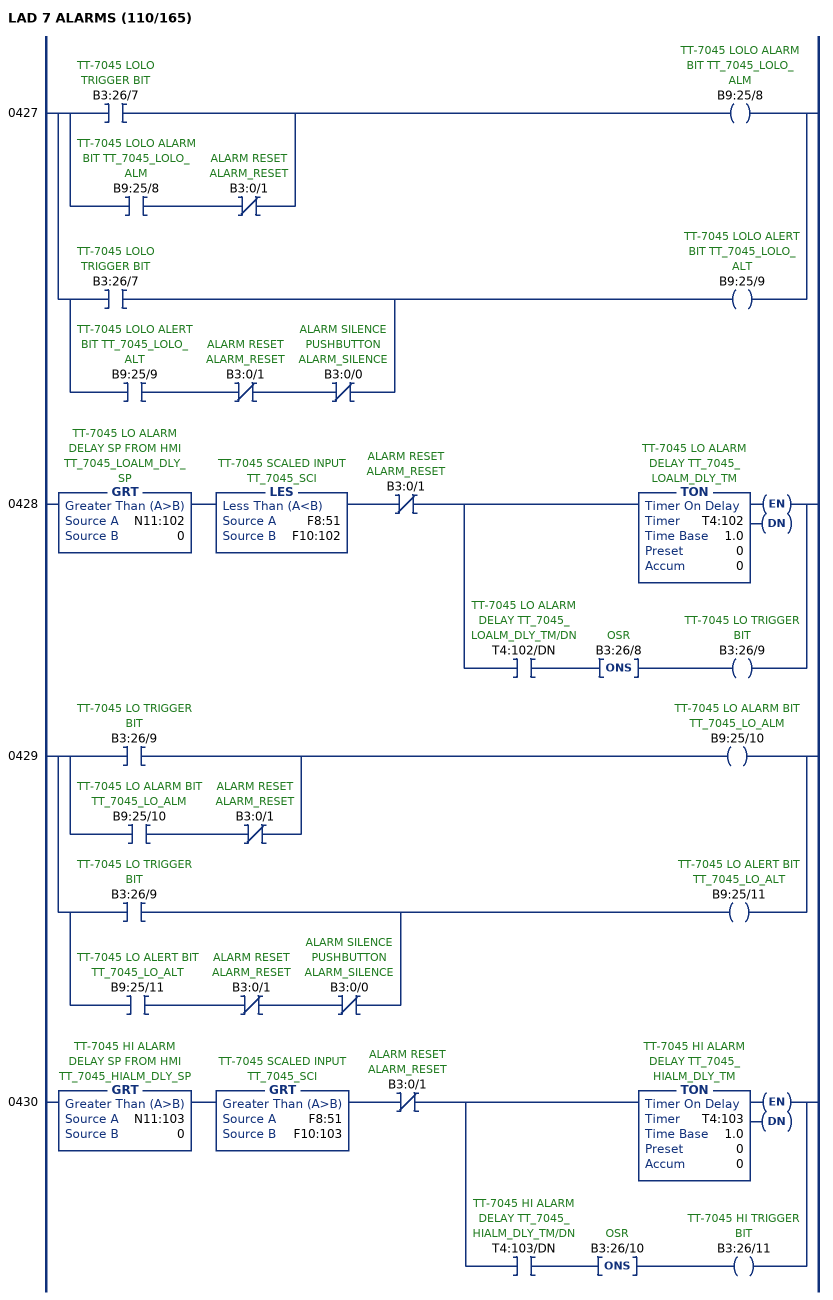
% Rung: 427 %
SOR BST BST XIC B3:26/7 NXB XIC B9:25/8 XIO B3:0/1 BND OTE B9:25/8 NXB BST XIC B3:26/7 NXB XIC B9:25/9 XIO B3:0/1 XIO B3:0/0 BND OTE B9:25/9 BND EOR
%   B3:26/7  "TT-7045 LOLO TRIGGER BIT" %
%   B9:25/8  TT_7045_LOLO_ALM  "TT-7045 LOLO ALARM BIT" %
%   B3:0/1  ALARM_RESET  "ALARM RESET" %
%   B9:25/9  TT_7045_LOLO_ALT  "TT-7045 LOLO ALERT BIT" %
%   B3:0/0  ALARM_SILENCE  "ALARM SILENCE PUSHBUTTON" %
% Rung: 428 %
SOR GRT N11:102 0 LES F8:51 F10:102 XIO B3:0/1 BST TON T4:102 1.0 0 0 NXB XIC T4:102/DN OSR B3:26/8 OTE B3:26/9 BND EOR
%   N11:102  TT_7045_LOALM_DLY_SP  "TT-7045 LO ALARM DELAY SP FROM HMI" %
%   F8:51  TT_7045_SCI  "TT-7045 SCALED INPUT" %
%   F10:102  TT_7045_LOALM_SP  "TT-7045 LO ALARM SP" %
%   B3:0/1  ALARM_RESET  "ALARM RESET" %
%   T4:102  TT_7045_LOALM_DLY_TM  "TT-7045 LO ALARM DELAY" %
%   B3:26/8  "OSR" %
%   B3:26/9  "TT-7045 LO TRIGGER BIT" %
% Rung: 429 %
SOR BST BST XIC B3:26/9 NXB XIC B9:25/10 XIO B3:0/1 BND OTE B9:25/10 NXB BST XIC B3:26/9 NXB XIC B9:25/11 XIO B3:0/1 XIO B3:0/0 BND OTE B9:25/11 BND EOR
%   B3:26/9  "TT-7045 LO TRIGGER BIT" %
%   B9:25/10  TT_7045_LO_ALM  "TT-7045 LO ALARM BIT" %
%   B3:0/1  ALARM_RESET  "ALARM RESET" %
%   B9:25/11  TT_7045_LO_ALT  "TT-7045 LO ALERT BIT" %
%   B3:0/0  ALARM_SILENCE  "ALARM SILENCE PUSHBUTTON" %
% Rung: 430 %
SOR GRT N11:103 0 GRT F8:51 F10:103 XIO B3:0/1 BST TON T4:103 1.0 0 0 NXB XIC T4:103/DN OSR B3:26/10 OTE B3:26/11 BND EOR
%   N11:103  TT_7045_HIALM_DLY_SP  "TT-7045 HI ALARM DELAY SP FROM HMI" %
%   F8:51  TT_7045_SCI  "TT-7045 SCALED INPUT" %
%   F10:103  TT_7045_HIALM_SP  "TT-7045 HI ALARM SP" %
%   B3:0/1  ALARM_RESET  "ALARM RESET" %
%   T4:103  TT_7045_HIALM_DLY_TM  "TT-7045 HI ALARM DELAY" %
%   B3:26/10  "OSR" %
%   B3:26/11  "TT-7045 HI TRIGGER BIT" %

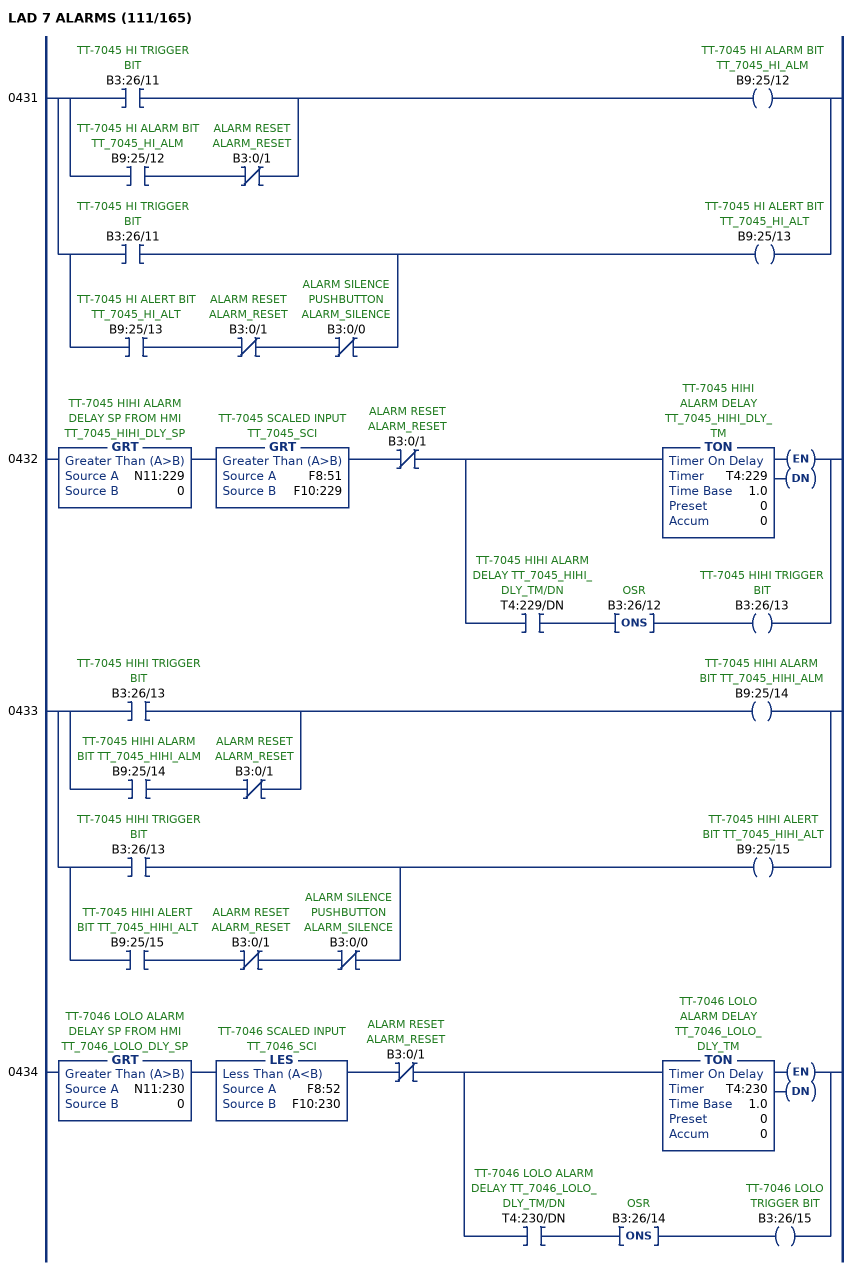
% Rung: 431 %
SOR BST BST XIC B3:26/11 NXB XIC B9:25/12 XIO B3:0/1 BND OTE B9:25/12 NXB BST XIC B3:26/11 NXB XIC B9:25/13 XIO B3:0/1 XIO B3:0/0 BND OTE B9:25/13 BND EOR
%   B3:26/11  "TT-7045 HI TRIGGER BIT" %
%   B9:25/12  TT_7045_HI_ALM  "TT-7045 HI ALARM BIT" %
%   B3:0/1  ALARM_RESET  "ALARM RESET" %
%   B9:25/13  TT_7045_HI_ALT  "TT-7045 HI ALERT BIT" %
%   B3:0/0  ALARM_SILENCE  "ALARM SILENCE PUSHBUTTON" %
% Rung: 432 %
SOR GRT N11:229 0 GRT F8:51 F10:229 XIO B3:0/1 BST TON T4:229 1.0 0 0 NXB XIC T4:229/DN OSR B3:26/12 OTE B3:26/13 BND EOR
%   N11:229  TT_7045_HIHI_DLY_SP  "TT-7045 HIHI ALARM DELAY SP FROM HMI" %
%   F8:51  TT_7045_SCI  "TT-7045 SCALED INPUT" %
%   F10:229  TT_7045_HIHI_SP  "TT-7045 HIHI ALARM SP" %
%   B3:0/1  ALARM_RESET  "ALARM RESET" %
%   T4:229  TT_7045_HIHI_DLY_TM  "TT-7045 HIHI ALARM DELAY" %
%   B3:26/12  "OSR" %
%   B3:26/13  "TT-7045 HIHI TRIGGER BIT" %
% Rung: 433 %
SOR BST BST XIC B3:26/13 NXB XIC B9:25/14 XIO B3:0/1 BND OTE B9:25/14 NXB BST XIC B3:26/13 NXB XIC B9:25/15 XIO B3:0/1 XIO B3:0/0 BND OTE B9:25/15 BND EOR
%   B3:26/13  "TT-7045 HIHI TRIGGER BIT" %
%   B9:25/14  TT_7045_HIHI_ALM  "TT-7045 HIHI ALARM BIT" %
%   B3:0/1  ALARM_RESET  "ALARM RESET" %
%   B9:25/15  TT_7045_HIHI_ALT  "TT-7045 HIHI ALERT BIT" %
%   B3:0/0  ALARM_SILENCE  "ALARM SILENCE PUSHBUTTON" %
% Rung: 434 %
SOR GRT N11:230 0 LES F8:52 F10:230 XIO B3:0/1 BST TON T4:230 1.0 0 0 NXB XIC T4:230/DN OSR B3:26/14 OTE B3:26/15 BND EOR
%   N11:230  TT_7046_LOLO_DLY_SP  "TT-7046 LOLO ALARM DELAY SP FROM HMI" %
%   F8:52  TT_7046_SCI  "TT-7046 SCALED INPUT" %
%   F10:230  TT_7046_LOLO_SP  "TT-7046 LOLO ALARM SP" %
%   B3:0/1  ALARM_RESET  "ALARM RESET" %
%   T4:230  TT_7046_LOLO_DLY_TM  "TT-7046 LOLO ALARM DELAY" %
%   B3:26/14  "OSR" %
%   B3:26/15  "TT-7046 LOLO TRIGGER BIT" %

